// TwinCAT 3 PLC project CamerasTCP_Drivers
// ProgramVersion: 3.1.4026.19
// libraries:
//   AI Codes And Validation, * (Marden Edwards)
//   Tc2_SerialCom, * (Beckhoff Automation GmbH)
//   Tc2_Standard, * (Beckhoff Automation GmbH)
//   Tc2_System, * (Beckhoff Automation GmbH)
//   Tc2_TcpIp, * (Beckhoff Automation GmbH)
//   Tc2_Utilities, * (Beckhoff Automation GmbH)
//   TcUnit, * (www.tcunit.org)
// project tree:
//   DUTs/ E_TCPIP_RequescCommand.TcDUT, E_TCPIP_SEND_STATE.TcDUT, E_TCPIP_StateWP.TcDUT
//   DUTs/METS/ADS Symobol/ E_SYMBOL_AccessState.TcDUT, E_SYMBOL_AdsStates.TcDUT, ST_SYMBOL_AddressInfo.TcDUT
//   DUTs/METS/AI Codes And Validation/ E_CodeAI.TcDUT, E_CodeAIType.TcDUT (not stored), E_CodeType.TcDUT, ST_CodeInfo.TcDUT, ST_CodeValidation.TcDUT, ST_RejectItems.TcDUT, ST_RejectReasonsForCase.TcDUT, ST_RejectReasonsForOuter.TcDUT, ST_RejectReasonsForPack.TcDUT
//   DUTs/METS/AI Codes And Validation/GS1_Standard/ E_GS1_CodeAIType.TcDUT, E_GS1_CodeLvl.TcDUT, ST_GS1_AI_Attributs.TcDUT, ST_GS1_AI_Definition.TcDUT, ST_GS1_CodeInfo.TcDUT, ST_GS1_CodeValidation.TcDUT, ST_GS1_Decode_AI.TcDUT
//   DUTs/METS/Alarms/ E_MessageID.TcDUT (not stored), E_MessageType.TcDUT, ST_AlarmDB.TcDUT, ST_Alarms.TcDUT, ST_AlarmSettings.TcDUT, ST_AlarmsTable.TcDUT, ST_AlarmStatus.TcDUT, ST_ALARM_Aux.TcDUT (not stored)
//   DUTs/METS/Aliases/ T_CAC_Filename.TcDUT, T_CASE_Barcode.TcDUT, T_Char.TcDUT, T_CHM_Filename.TcDUT, T_CodeBATCH.TcDUT, T_CodeBRAND.TcDUT, T_CodeCRYPTO.TcDUT, T_CodeGTIN.TcDUT, T_CodeMRP.TcDUT, T_CodePIT.TcDUT, T_CodePO.TcDUT, T_CodePRODUCEDATE.TcDUT, T_CodeRSKU.TcDUT, T_CodeURL.TcDUT, T_DB_LongSTRING.TcDUT, T_FileExtension.TcDUT, T_FolderName.TcDUT, T_FolderPath.TcDUT, T_FSS_RejecCode.TcDUT, T_HMI_PACK_Barcode.TcDUT, T_ISO8601Time.TcDUT, T_LongSTRING.TcDUT, T_OAC_Filename.TcDUT, T_OCV_Filename.TcDUT, T_OHM_Filename.TcDUT, T_OUTER_Barcode.TcDUT, T_PACK_Barcode.TcDUT, T_PCM_Filename.TcDUT, T_PositiveDINT.TcDUT, T_PositiveINT.TcDUT, T_ProductDescription.TcDUT, T_RejectCode.TcDUT, T_TimeLog.TcDUT
//   DUTs/METS/Case/CAC/ E_CAC_State.TcDUT, ST_CAC_Data.TcDUT
//   DUTs/METS/Case/CHM/CHM Data Structure/GenericHierarchy/Case Item Structures/ ST_CaseContent.TcDUT, ST_CaseIdentity.TcDUT, ST_CaseItem.TcDUT
//   DUTs/METS/Case/CHM/CHM Data Structure/GenericHierarchy/Outer Item Structures/ ST_OuterContent.TcDUT, ST_OuterIdentity.TcDUT, ST_OuterItem.TcDUT
//   DUTs/METS/Case/CHM/CHM Data Structure/GenericHierarchy/Pack Item Structures/ ST_PackIdentity.TcDUT, ST_PackItem.TcDUT
//   DUTs/METS/Case/CHM/CHM Data Structure/GenericHierarchy/ ST_DefaultIdentity.TcDUT
//   DUTs/METS/Case/CHM/CHM Data Structure/ ST_Attributes.TcDUT, ST_CHM_GenericHierarchy.TcDUT (excluded from build), ST_GenericHierarchy.TcDUT, ST_MessageHeader.TcDUT
//   DUTs/METS/Case/CHM/ E_CHM_GeneratorState.TcDUT, E_CHM_State.TcDUT, E_CHM_WriteMode.TcDUT (excluded from build), ST_CHM_Data.TcDUT
//   DUTs/METS/Case/ E_CASE_State.TcDUT, ST_CasePackerInfo.TcDUT, ST_CASE_CaseQueue.TcDUT, ST_CASE_DefferOuter.TcDUT, ST_CASE_InfeedQueue.TcDUT, ST_CASE_OperationData.TcDUT (not stored)
//   DUTs/METS/Case/ORCA/ E_ORCA_State.TcDUT, ST_ORCA_BrandInfo.TcDUT, ST_ORCA_Data.TcDUT, ST_ORCA_Outers.TcDUT, ST_ORCA_ProductInfo.TcDUT, ST_ORCA_SiteInfo.TcDUT
//   DUTs/METS/Device/CX Unit/Device/ E_CX_DeviceState.TcDUT
//   DUTs/METS/Device/CX Unit/EtherCAT/ E_CX_EtherCATState.TcDUT (not stored), ST_CX_EtherCATDeviceState.TcDUT, ST_CX_EtherCATMasterPNetState.TcDUT, ST_CX_EtherCATMasterState.TcDUT
//   DUTs/METS/Device/CX Unit/EtherCAT/Terminal FBs/EBUS/ ST_EBUS_AnalogueDataIn.TcDUT, ST_EBUS_EtherCATState.TcDUT
//   DUTs/METS/Device/CX Unit/EtherCAT/Terminal FBs/KBUS/ E_KBUS_RegisterAccessState.TcDUT, ST_KBUS_AnalogueDataIn.TcDUT, ST_KBUS_AnalogueDataOut.TcDUT, ST_KBUS_KL1501DataIn.TcDUT, ST_KBUS_KL1501DataOut.TcDUT, ST_KBUS_KL5001Config.TcDUT
//   DUTs/METS/Device/CX Unit/EtherCAT/Terminal FBs/ ST_EtherCATSlaveInfo.TcDUT, ST_EtherCATStatus.TcDUT
//   DUTs/METS/Device/CX Unit/Network/ E_CX_NetworkInfoState.TcDUT, E_CX_SetAMSNetIDState.TcDUT, ST_CX_AdapterInfo.TcDUT, ST_CX_NetworkInfo.TcDUT
//   DUTs/METS/Device/CX Unit/NOVRAM/ E_CX_NVDataCtrlState.TcDUT, E_CX_NVDataOpMode.TcDUT (not stored), E_CX_NVXMLState.TcDUT (not stored), ST_CX_AMSAddress.TcDUT, ST_CX_EL6080DataIn.TcDUT, ST_CX_EL6080DataOut.TcDUT, ST_CX_NVDataBlock.TcDUT
//   DUTs/METS/Device/CX Unit/System/ E_CX_HWType.TcDUT, E_CX_State.TcDUT (not stored)
//   DUTs/METS/Device/Cylinders/ E_CYLINDER_Name.TcDUT (not stored), E_CYLINDER_Position.TcDUT, ST_CYLINDER_Config.TcDUT (not stored), ST_CYLINDER_Control.TcDUT, ST_CYLINDER_IN.TcDUT, ST_CYLINDER_OUT.TcDUT, ST_CYLINDER_Status.TcDUT, ST_CYLINDER_TagID.TcDUT
//   DUTs/METS/Device/DB/ E_DB_ScanState.TcDUT (not stored), ST_DB_CACDataCtrl.TcDUT (not stored), ST_DB_OACDataCtrl.TcDUT, ST_DB_OCVDataCtrl.TcDUT
//   DUTs/METS/Device/DB/OLD/ ST_DBResult.TcDUT (excluded from build), ST_DB_CACCheckCtrl.TcDUT (excluded from build), ST_DB_Config.TcDUT, ST_DB_OACCheckCtrl.TcDUT (excluded from build), ST_DB_OCVCheckCtrl.TcDUT (excluded from build), ST_DB_PcvCheckCtrl.TcDUT (excluded from build), ST_DB_ReportDBCtrl.TcDUT, ST_DB_ReportResult.TcDUT
//   DUTs/METS/Device/Drive/Analog/Config/ ST_AnalogDrive.TcDUT
//   DUTs/METS/Device/Drive/Analog/ ST_DriveCtrl.TcDUT, ST_PhtcCtrl.TcDUT (excluded from build)
//   DUTs/METS/Device/Drive/MC2/Axis Control/ E_AXIS_MotionType.TcDUT (not stored), ST_AXIS_Control.TcDUT, ST_AXIS_IN.TcDUT, ST_AXIS_OUT.TcDUT, ST_AXIS_Status.TcDUT
//   DUTs/METS/Device/Drive/MC2/Config/ ST_AXIS_Config.TcDUT
//   DUTs/METS/Device/Drive/MC2/EtherCAT/AX5000 FBs/ ST_AX5000_TouchProbe.TcDUT
//   DUTs/METS/Device/Drive/MC2/EtherCAT/Encoder FBs/ ST_DeviceAddress.TcDUT
//   DUTs/METS/Device/Drive/MC2/ E_MC_Name.TcDUT (not stored)
//   DUTs/METS/Device/Drive/MC2/NC Axis/Cam/ E_CAM_Update.TcDUT (not stored)
//   DUTs/METS/Device/Drive/MC2/NC Axis/ E_AXIS_CtrlState.TcDUT, E_TORQUE_Scaling.TcDUT, ST_AxisCtrlRamps.TcDUT, ST_DriveStatus.TcDUT, ST_LatchPosBuffer.TcDUT, ST_NC_EncDataIn.TcDUT, ST_NC_EncDataOut.TcDUT
//   DUTs/METS/Device/Drive/MC2/TempAxis/ ST_AxisHomeStruct.TcDUT (excluded from build), ST_AxisMotionStruct.TcDUT (excluded from build)
//   DUTs/METS/Device/Drive/Profinet/Config/ ST_ProfinetDrive.TcDUT, ST_ProfinetMasterConfig.TcDUT
//   DUTs/METS/Device/Drive/Profinet/ E_DRIVE_Name.TcDUT, ST_PNetMasterStatus.TcDUT
//   DUTs/METS/Device/Drive/Profinet/Parameters/ ST_DataPntAdr.TcDUT, ST_KeyPadDisplay.TcDUT, ST_Parameter.TcDUT, ST_ParameterControl.TcDUT, ST_Parameters.TcDUT, ST_Value.TcDUT
//   DUTs/METS/Device/Drive/Profinet/_G120/Drives/ E_DRIVE_DataType.TcDUT, ST_DRIVE_INPUT.TcDUT, ST_DRIVE_OUTPUT.TcDUT, ST_DRIVE_STATUS.TcDUT, ST_G120_ExtendedIn.TcDUT, ST_G120_ExtendedOut.TcDUT, ST_G120_IN.TcDUT, ST_G120_OUT.TcDUT (not stored), ST_G120_Status.TcDUT
//   DUTs/METS/Device/Drive/Profinet/_G120/ ST_G120_Control.TcDUT
//   DUTs/METS/Device/Encoders/CAMS/ ST_AFS60_Cam.TcDUT, ST_AFS60_CamHMi.TcDUT, ST_AFS60_Config.TcDUT, ST_AFS60_Status.TcDUT
//   DUTs/METS/Device/Encoders/ E_ENOCDER_Name.TcDUT (not stored), ST_ENCODER_IN.TcDUT, ST_ENCODER_OUT.TcDUT, ST_ENCODER_Status.TcDUT
//   DUTs/METS/Device/IO2 Controls/ E_IO2_InputSource.TcDUT, E_IO2_Type.TcDUT, ST_IO2_Diagnostic.TcDUT, ST_IO2_InputPLC.TcDUT, ST_IO2_OutputPLC.TcDUT
//   DUTs/METS/Device/IO2 Controls/Input Ctrl/ ST_IO2_DoubleInputCtrl.TcDUT, ST_IO2_DoubleInputLockedCtrl.TcDUT, ST_IO2_SingleInputCtrl.TcDUT, ST_IO2_SingleInputLockedCtrl.TcDUT
//   DUTs/METS/Device/IO2 Controls/Outpout Ctrl/ ST_IO2_OutputCtrl.TcDUT
//   DUTs/METS/Device/Printers/ E_PRINTER_Name.TcDUT (not stored), E_PRINTER_State.TcDUT, ST_PRINTER_Config.TcDUT, ST_PRINTER_IN.TcDUT, ST_PRINTER_OUT.TcDUT, ST_PRINTER_Status.TcDUT
//   DUTs/METS/Device/Scanner/ E_ClientSteps.TcDUT (not stored), E_DataExchaSteps.TcDUT (not stored), E_SCANNER_CodeType.TcDUT, E_SCANNER_DeviceType.TcDUT, E_SCANNER_Name.TcDUT (not stored), E_SCANNER_State.TcDUT, E_SCANNER_Vendor.TcDUT, ST_SCANNER.TcDUT, ST_SCANNER_ApplicationIdentifier.TcDUT, ST_SCANNER_CameraMap.TcDUT, ST_SCANNER_CodeData.TcDUT, ST_SCANNER_Config.TcDUT, ST_SCANNER_Evaluation.TcDUT, ST_SCANNER_ImageData.TcDUT, ST_SCANNER_ManualCtrl.TcDUT, ST_SCANNER_OpState.TcDUT, ST_SCANNER_Options.TcDUT, ST_SCANNER_Performance.TcDUT, ST_SCANNER_Statistics.TcDUT, ST_SCANNER_TriggerID.TcDUT
//   DUTs/METS/Device/Scanner/Hand Scanner/ E_ConnectSteps.TcDUT (not stored), E_DataSequence.TcDUT, E_SCANNER_Baudrate.TcDUT (not stored), ST_SCANNER_HoneywellConfig.TcDUT, ST_SCANNER_HoneywellCtrl.TcDUT, ST_SCANNER_HoneywellStatus.TcDUT, ST_SCANNER_HostAck.TcDUT, ST_SCANNER_USBConfig.TcDUT
//   DUTs/METS/Device/Scanner/NewModel/ ST_SCANNER_Configuration.TcDUT (not stored), ST_SCANNER_Ctrl.TcDUT, ST_SCANNER_CtrlMapping.TcDUT (not stored), ST_SCANNER_CtrlOptions.TcDUT (excluded from build), ST_SCANNER_IN.TcDUT, ST_SCANNER_ManualStatus.TcDUT (not stored), ST_SCANNER_OUT.TcDUT (not stored), ST_SCANNER_Status.TcDUT (not stored)
//   DUTs/METS/Files/ E_FILE_CtrlState.TcDUT, E_FILE_DeleteOldFilesState.TcDUT, E_FILE_State.TcDUT, ST_FILE_WriteFileStatistic.TcDUT
//   DUTs/METS/HMI/Device Manual Control/ ST_HMI_AxisCtrl.TcDUT, ST_HMI_CylinderCtrl.TcDUT (not stored), ST_HMI_G120Ctrl.TcDUT, ST_HMI_PrinterCtrl.TcDUT
//   DUTs/METS/HMI/Device Status/ E_HMI_DriveStatus.TcDUT, ST_HMI_AxisStatus.TcDUT, ST_HMI_CylinderStatus.TcDUT, ST_HMI_G120Status.TcDUT (not stored), ST_HMI_HoneywellStatus.TcDUT, ST_HMI_PrinterStatus.TcDUT
//   DUTs/METS/HMI/HMIQueue/ ST_HMI_CAC_Data.TcDUT, ST_HMI_CaseRejectCode.TcDUT (not stored), ST_HMI_CaseVerifiedCode.TcDUT, ST_HMI_CASE_CaseQueue.TcDUT, ST_HMI_InfeedQueue.TcDUT (not stored), ST_HMI_OAC_Data.TcDUT, ST_HMI_OCV_Data.TcDUT, ST_HMI_OuterStatus.TcDUT, ST_HMI_PACK_BufferStatus.TcDUT (not stored), ST_HMI_PLAS_Queue.TcDUT
//   DUTs/METS/HMI/ ST_HMI_BarGraph.TcDUT (not stored), ST_HMI_Buttons.TcDUT, ST_HMI_CSVStoreTable.TcDUT (not stored), ST_HMI_StationStatus.TcDUT, ST_HMI_Visualisation.TcDUT
//   DUTs/METS/KPI/ ST_KPI_CasePackerSignals.TcDUT, ST_KPI_CodePos.TcDUT, ST_KPI_InspectionEfficency.TcDUT, ST_KPI_ItemsProduced.TcDUT, ST_KPI_OCVFile.TcDUT, ST_KPI_OutersProcessing.TcDUT, ST_KPI_OutersProduced.TcDUT
//   DUTs/METS/LogData/ E_LOG_Handler.TcDUT, ST_LOG_Alarms.TcDUT, ST_LOG_EventData.TcDUT, ST_LOG_FileWriteError.TcDUT, ST_LOG_MachineState.TcDUT, ST_LOG_RejectReasons.TcDUT (not stored), ST_LOG_WriteImageData.TcDUT
//   DUTs/METS/NV Data/ ST_NOVRAM_METS_Cameras.TcDUT, ST_NOVRAM_METS_CaseInspactionLog.TcDUT, ST_NOVRAM_METS_DualInputs.TcDUT, ST_NOVRAM_METS_EventCounters.TcDUT (not stored), ST_NOVRAM_METS_Inspection.TcDUT
//   DUTs/METS/Outers/ E_OUTER_AgrregationState.TcDUT, E_OUTER_State.TcDUT, ST_OUTER_Status.TcDUT
//   DUTs/METS/Outers/OAC/ E_OAC_State.TcDUT, ST_OAC_Data.TcDUT
//   DUTs/METS/Outers/SFLX/ E_SIDEFLEX_UnitType.TcDUT, ST_SIDEFLEX_Offset.TcDUT, ST_SIDEFLEX_ProcessData.TcDUT
//   DUTs/METS/Packs/ E_OCV_CheckMode.TcDUT, E_OCV_State.TcDUT, E_PACK_FilledInStatus.TcDUT, E_PACK_ReadStep.TcDUT, E_PACK_State.TcDUT, ST_PACK_CodeBuffer.TcDUT, ST_PACK_CodeStatus.TcDUT, ST_PACK_ConfirmationQueue.TcDUT, ST_PACK_Data.TcDUT, ST_PACK_DuplicatesCheck.TcDUT (not stored), ST_PACK_InfeedQueue.TcDUT, ST_PACK_InTransferQueue.TcDUT, ST_PACK_LastFilledCodes.TcDUT (not stored), ST_PACK_TriggerOffset.TcDUT
//   DUTs/METS/Packs/_Lab/ ST_LAB_OuterData_1.TcDUT, ST_LAB_PackData_1.TcDUT
//   DUTs/METS/PCM/ E_PCM_State.TcDUT (not stored), ST_PCM_Data.TcDUT (not stored), ST_PCM_Status.TcDUT
//   DUTs/METS/PCM/PCM_Hierarchy/ProductInformation/Product/ ST_HierarchyData.TcDUT, ST_HierarchyDataList.TcDUT (not stored)
//   DUTs/METS/PCM/PCM_Hierarchy/ProductInformation/Settings/ ST_ToleranceThresholdCS.TcDUT, ST_ToleranceThresholdOUT.TcDUT, ST_ToleranceThresholdPK.TcDUT (not stored)
//   DUTs/METS/PCM/PCM_Hierarchy/ProductInformation/ ST_PCMProduct.TcDUT (not stored), ST_PCMSettings.TcDUT (not stored)
//   DUTs/METS/PCM/PCM_Hierarchy/ ST_PCMMessageHeader.TcDUT (not stored), ST_ProductInformation.TcDUT (not stored)
//   DUTs/METS/String Processing/ E_STRING_ExtrMode.TcDUT (not stored)
//   DUTs/METS/System/ E_SYSTEM_CTState.TcDUT, E_SYSTEM_HandScannerBaudrate.TcDUT, E_SYSTEM_ItemType.TcDUT, E_SYSTEM_MachineState.TcDUT, E_SYSTEM_MaintainFolders.TcDUT, E_SYSTEM_OSType.TcDUT, ST_SYSTEM_Config.TcDUT, ST_SYSTEM_DateTime.TcDUT, ST_SYSTEM_DeviceState.TcDUT, ST_SYSTEM_Door.TcDUT, ST_SYSTEM_MachineID.TcDUT (not stored), ST_SYSTEM_MachineMode.TcDUT, ST_SYSTEM_MachineState.TcDUT, ST_SYSTEM_ProductionLine.TcDUT, ST_SYSTEM_SafetyStatus.TcDUT, ST_SYSTEM_SoftwareVersion.TcDUT
//   DUTs/METS/System/Status/ ST_SYSTEM_ArchiveDBStatus.TcDUT (not stored), ST_SYSTEM_BridgeStatus.TcDUT, ST_SYSTEM_LoggerStatus.TcDUT (not stored), ST_SYSTEM_MachineStatus.TcDUT, ST_SYSTEM_ReportingDBStatus.TcDUT
//   DUTs/METS/System/System Modes/ E_SYSTEM_AutomationMode.TcDUT (not stored), E_SYSTEM_OuterAggregationMode.TcDUT (not stored), E_SYSTEM_PackAggregationMode.TcDUT
//   DUTs/METS/TCPIP Address/ E_TCPIP_State_1.TcDUT, ST_TCPIP_AddressPort.TcDUT
//   DUTs/METS/XML Processing/ E_XML_CtrlState.TcDUT, E_XML_GeneratorState.TcDUT, E_XML_WritingMode.TcDUT
//   DUTs/METS/_StationOperational/C715 Tempalate Example/ E_04_ElevatorState_C715.TcDUT, E_Axis_C715.TcDUT, E_Cylinder_C715.TcDUT, ST_04_ElevatorSeq_C715.TcDUT, ST_BundleTrackingRegister_C715.TcDUT, ST_CommonStationConfig_C715.TcDUT (not stored)
//   DUTs/METS/_StationOperational/ E_00_StationStateTemplate.TcDUT, ST_00_StationStructTemplate.TcDUT
//   DUTs/METS/_StationOperational/Manual Machine/ E_OuterPrintStationState.TcDUT, ST_OuterPrintStationStruct.TcDUT
//   DUTs/METS/_StationOperational/SeqCtrl/ ST_STATION_Requests.TcDUT, ST_STATION_Status.TcDUT
//   DUTs/Test_DUTs/ ST_DuplicateInfo.TcDUT, ST_FBinside.TcDUT, ST_LAB_CaseData.TcDUT, ST_LAB_OuterData.TcDUT, ST_LAB_PackData.TcDUT
//   GVLs/ CodeAI.TcGVL, gConstants.TcGVL, GVL.TcGVL, GVL_HIKROBOT_COMMANDS.TcGVL, GVL_test.TcGVL
//   / PlcTask.TcTTO, TcUnit_Task.TcTTO
//   POUs/FBReferenceTest/ FB_TimersTEST.TcPOU, PRG_Reference_POU.TcPOU
//   POUs/FinaliseCaseData/ FB_CASE_DuplicatCheck.TcPOU, FB_CASE_DuplicateUpdateToDB.TcPOU, FB_CASE_FinaliseData.TcPOU, FB_CASE_InitialiseData.TcPOU, FB_CASE_MovePackerToCase.TcPOU, FB_CASE_ValidateContent.TcPOU
//   POUs/ PRG_TEST.TcPOU
//   POUs/TcUnit/FB_CASE_DuplicatCheckTests/ FB_CASE_DuplicatCheckTests.TcPOU, PRG_CASE_DuplicatCheckManual.TcPOU
//   POUs/TcUnit/FB_CASE_DuplicateUpdateToDBTests/ PRG_CASE_DuplicateUpdateToDBManual.TcPOU, FB_CASE_DuplicateUpdateToDBTests.TcPOU
//   POUs/TcUnit/FB_CASE_ValidateContentTests/ FB_CASE_ValidateContentTests.TcPOU, PRG_CASE_ValidateContentManual.TcPOU
//   POUs/TcUnit/FB_CASE_InitialiseData/ FB_CASE_InitialiseDataTests.TcPOU, PRG_CASE_InitialiseDataManual.TcPOU
//   POUs/TcUnit/FB_CASE_FinaliseDataTests/ FB_CASE_FinaliseDataTests.TcPOU, PRG_CASE_FinaliseDataManual.TcPOU
//   POUs/TcUnit/F_CODE_GetItemAITests/ PRG_CODE_GetItemAIManual.TcPOU
//   POUs/_Utilites/Addtionals/ FB_PulseGenerator_Sync.TcPOU, PRG_ButtonsHandler.TcPOU
//   POUs/_Utilites/CAMERAS/ FB_SCANNER_HikrobotEXT.TcPOU, F_CREATE_MESSAGE.TcPOU
//   POUs/_Utilites/METS/Common LIB/08_SOFTWARE LIB/AI Codes And Validation FBs/ FB_CODE_ClearCodeInfo.TcPOU, FB_CODE_ValidateExplicitCode.TcPOU (not stored), F_CODE_AssignValToStringWithPrefix.TcPOU, F_CODE_GetItemAI.TcPOU (not stored)
//   POUs/_Utilites/METS/Common LIB/08_SOFTWARE LIB/AI GS1 Codes And Validation FBs/ FB_GS1_ClearCodeInfo.TcPOU, FB_GS1_ValidateExplicitCode.TcPOU, F_GS1_GetItem.TcPOU
//   POUs/_Utilites/METS/Concat Function/ F_CONCAT3.TcPOU, F_CONCAT4.TcPOU, F_CONCAT5.TcPOU, F_CONCAT6.TcPOU, F_CONCAT7.TcPOU, F_CONCAT8.TcPOU, F_CONCAT9.TcPOU
//   POUs/_Utilites/METS/ FB_ExtractString.TcPOU (not stored), F_CASE_GetSKUFromHex.TcPOU, F_CODE_BATSerializator.TcPOU (not stored), F_CODE_GetItem.TcPOU, F_FiltredSetBitState16.TcPOU, F_InvalidateASCIIChar.TcPOU, F_SafeDIV.TcPOU, F_StringAddPrefix.TcPOU (not stored), F_StringWildcard.TcPOU, F_SYSTEM_SystemTimeAsISO8601.TcPOU, F_SYSTEM_SystemTimeOffsetToHHMM.TcPOU, F_ZeroPadString.TcPOU
//   POUs/_Utilites/TCP_FB/ FB_ReceiveString.TcPOU, FB_TCP_ClientPortCtrl.TcPOU
//   POUs/_Utilites/Tests/ FB_FIND_OuterDuplicates.TcPOU, FB_FIND_OuterDuplicatesPiotr.TcPOU, FB_FIND_OuterDuplicatesPiotrAI.TcPOU, IO_logic.TcPOU, Outer_IN_Case_Duplicat.TcPOU, PRG_TestCamera.TcPOU

CONFIGURATION CamerasTCP_Drivers
    RESOURCE PLC ON TwinCAT3
        TASK PlcTask(INTERVAL := T#20ms, PRIORITY := 20);
        TASK TcUnit_Task(INTERVAL := T#1ms, PRIORITY := 25);
        PROGRAM PRG_TEST WITH TcUnit_Task : PRG_TEST;
    END_RESOURCE
END_CONFIGURATION

// ---- DUTs/E_TCPIP_RequescCommand.TcDUT
{attribute 'qualified_only'}
{attribute 'strict'}
{attribute 'to_string'}
TYPE E_TCPIP_RequescCommand :
(
	NONE,					(* No request to send *)
	SetRunMode,				(* Set run mode, 0 - Normal, 1 - Raw, 2 - Test *)
	SetAcq,					(* Set acquisition mode, 0 - Stop acq, 1 - Start acq *)
	GetUserCur,
	HeartbeatCheck,		
	SetAquisitonModeON,
	SetAquisitionModeOFF,
	WrongReply	
);
END_TYPE

// ---- DUTs/E_TCPIP_SEND_STATE.TcDUT
{attribute 'qualified_only'}
{attribute 'strict'}
{attribute 'to_string'}
TYPE E_TCPIP_SEND_STATE :
(
	WAITING,
	SEND,
	RECEIVE,
	DONE,
	CONN_RESET,
	HEARTBEAT_CHECK
);
END_TYPE

// ---- DUTs/E_TCPIP_StateWP.TcDUT
{attribute 'qualified_only'}
{attribute 'strict'}
{attribute 'to_string'}
TYPE E_TCPIP_StateWP :
(
	E_TCPIP_IDLE,
	E_TCPIP_CONNECT,
	E_TCPIP_SEND,
	E_TCPIP_RECEIVE,
	E_TCPIP_DISCONNECT,
	E_TCPIP_CLOSEALL,
	E_TCPIP_DONE
);
END_TYPE

// ---- DUTs/METS/ADS Symobol/E_SYMBOL_AccessState.TcDUT
TYPE E_SYMBOL_AccessState :
(
	E_SYMBOL_IDLE,
	E_SYMBOL_GETSYMBOLINFO,
	E_SYMBOL_READDATA,
	E_SYMBOL_WRITEDATA,
	E_SYMBOL_DONE
);
END_TYPE

// ---- DUTs/METS/ADS Symobol/E_SYMBOL_AdsStates.TcDUT
TYPE E_SYMBOL_AdsStates :
(
	ADSSTATES_INVALID :=0,
	ADSSTATES_IDLE :=1,
	ADSSTATES_RESET :=2,
	ADSSTATES_INIT :=3,
	ADSSTATES_START :=4,
	ADSSTATES_RUN :=5,
	ADSSTATES_STOP :=6,
	ADSSTATES_SAVECFG :=7,
	ADSSTATES_LOADCFG :=8,
	ADSSTATES_POWERFAILURE :=9,
	ADSSTATES_POWERGOOD :=10,
	ADSSTATES_ERROR :=11
);
END_TYPE

// ---- DUTs/METS/ADS Symobol/ST_SYMBOL_AddressInfo.TcDUT
TYPE ST_SYMBOL_AddressInfo :	(* 8 bytes *)
STRUCT
	pSymAddr	: 	DWORD;
	nSymSize	:	UDINT;
END_STRUCT
END_TYPE

// ---- DUTs/METS/AI Codes And Validation/E_CodeAI.TcDUT
{attribute 'qualified_only'}
TYPE E_CodeAI :
(
	GTIN 			:= 1,
	BATCH 			:= 10,
	SERIAL			:= 21,
	PO				:= 91,
	BRANDSPEC		:= 92,
	CRYPTO			:= 93,
	PRODDATE		:= 94,
	RSKU 			:= 240,
	MRP				:= 8005,
	USERFIELD		:= 999
);
END_TYPE

// ---- DUTs/METS/AI Codes And Validation/E_CodeType.TcDUT
TYPE E_CodeType :
(
	E_NONE,
	E_PACK,
	E_INTERIM,
	E_OUTER,
	E_CASE

);
END_TYPE

// ---- DUTs/METS/AI Codes And Validation/GS1_Standard/E_GS1_CodeAIType.TcDUT
TYPE E_GS1_CodeAIType :
(
	GS1_00		:= 0,		(*GS1 Not defined*)
	GS1_01		 :=1,		(***********Global Trade Item Number (GTIN)	N2+N14*************)
	GS1_10		:=10,		(***********Batch or lot number	N2+X..20*************)
	GS1_11		:=11,		(***********Production date (YYMMDD)		N2+N6*************)
	GS1_15		:=15,		(***********Best before date (YYMMDD)			N2+N6*************)
	GS1_17		:=17,		(***********Expiration date (YYMMDD)		N2+N6*************)
	GS1_21		:=21,		(***********Serial number		N2+X..20*************)
	GS1_240		:=240,	(***********Additional product identification assigned by the manufacturer	N3+X..30*************)
	GS1_8005		:=8005,	(***********Price per unit of measure	N4+N6*************)
	GS1_8006		:=8006,	(***********Identification of an individual trade item piece	N4+N14+N2+N2*************)
	GS1_8008		:=8008,	(***********Date and time of production		N4+N8+N..4*************)
	GS1_91		:=91,		(***********Company internal information	N2+X..90*************)
	GS1_92		:=92,		(***********Company internal information	N2+X..90*************)
	GS1_93		:=93,		(***********Company internal information	N2+X..90*************)
	GS1_94		:=94,		(***********Company internal information	N2+X..90*************)
	NON_GS1_01		:=10001,	(***********Non GS1 - user defined		X..255*************)
	NON_GS1_02		:=10002,	(***********Non GS1 - user defined		X..255*************)
	NON_GS1_03		:=10003,	(***********Non GS1 - user defined		X..255*************)
	NON_GS1_04		:=10004,	(***********Non GS1 - user defined		X..255*************)
	NON_GS1_05		:=10005,	(***********Non GS1 - user defined		X..255*************)
	NON_GS1_06		:=10006,	(***********Non GS1 - user defined		X..255*************)
	NON_GS1_07		:=10007,	(***********Non GS1 - user defined		X..255*************)
	NON_GS1_08		:=10008,	(***********Non GS1 - user defined		X..255*************)
	NON_GS1_09		:=10009,	(***********Non GS1 - user defined		X..255*************)
	NON_GS1_10		:=10010	(***********Non GS1 - user defined		X..255*************)
);
END_TYPE

// ---- DUTs/METS/AI Codes And Validation/GS1_Standard/E_GS1_CodeLvl.TcDUT
TYPE E_GS1_CodeLvl :
(
	E_LVL_NONE,
	E_LEVEL1,
	E_LEVEL2,
	E_LEVEL3
);
END_TYPE

// ---- DUTs/METS/AI Codes And Validation/GS1_Standard/ST_GS1_AI_Attributs.TcDUT
TYPE ST_GS1_AI_Attributs :
STRUCT
	sDataField 	: T_MaxString;
	bDataChanged	: BOOL;
	sAI_Id		: STRING(5);
	eGS1_AI		: E_GS1_CodeAIType;
	bFixed		: BOOL;
	nLength		: UINT;
END_STRUCT
END_TYPE

// ---- DUTs/METS/AI Codes And Validation/GS1_Standard/ST_GS1_AI_Definition.TcDUT
TYPE ST_GS1_AI_Definition :
STRUCT
	sDotCode_CI	: STRING(3) := ']j';			(* GS1 marker (FNC1 Carrier Identifiers for DataMatrix barcode *)
	sDMC_CI		: STRING(3) := ']d2';			(* GS1 marker (FNC1 Carrier Identifiers for DataMatrix barcode *)
	sCode128_CI	: STRING(3) := ']c1';			(* GS1 marker (FNC1 Carrier Identifiers for Code128 barcode *)
	stAI_01_Lvl1	: ST_GS1_AI_Attributs := (sAI_Id:='01', eGS1_AI:=GS1_01, bFixed:= TRUE, nLength:=14);	(***********N2+N14*************)
	stAI_01_Lvl2	: ST_GS1_AI_Attributs := (sAI_Id:='01', eGS1_AI:=GS1_01, bFixed:= TRUE, nLength:=14);	(***********N2+N14*************)
	stAI_01_Lvl3	: ST_GS1_AI_Attributs := (sAI_Id:='01', eGS1_AI:=GS1_01, bFixed:= TRUE, nLength:=14);	(***********N2+N14*************)
	stAI_10		: ST_GS1_AI_Attributs := (sAI_Id:='10', eGS1_AI:=GS1_10, bFixed:= FALSE, nLength:=20);	(***********N2+X..20*************)
	stAI_11		: ST_GS1_AI_Attributs := (sAI_Id:='11', eGS1_AI:=GS1_11, bFixed:= TRUE, nLength:=6);	(***********N2+N6*************)
	stAI_15		: ST_GS1_AI_Attributs := (sAI_Id:='15', eGS1_AI:=GS1_15, bFixed:= TRUE, nLength:=6);	(***********N2+N6*************)
	stAI_17		: ST_GS1_AI_Attributs := (sAI_Id:='17', eGS1_AI:=GS1_17, bFixed:= TRUE, nLength:=6);	(***********N2+N6*************)
	stAI_21		: ST_GS1_AI_Attributs := (sAI_Id:='21', eGS1_AI:=GS1_21, bFixed:= FALSE, nLength:=20);	(***********N2+X..20*************)
	stAI_240		: ST_GS1_AI_Attributs := (sAI_Id:='240', eGS1_AI:=GS1_240, bFixed:= FALSE, nLength:=30);		(***********N3+X..30*************)
	stAI_8005		: ST_GS1_AI_Attributs := (sAI_Id:='8005', eGS1_AI:=GS1_8005, bFixed:= TRUE, nLength:=6);		(***********N4+N6*************)
	stAI_8006		: ST_GS1_AI_Attributs := (sAI_Id:='8006', eGS1_AI:=GS1_8006, bFixed:= TRUE, nLength:=18);	(***********N4+N14+N2+N2*************)
	stAI_8008		: ST_GS1_AI_Attributs := (sAI_Id:='8008', eGS1_AI:=GS1_8008, bFixed:= TRUE, nLength:=12);	(***********N4+N8+N..4*************)
	stAI_91		: ST_GS1_AI_Attributs := (sAI_Id:='91', eGS1_AI:=GS1_91, bFixed:= FALSE, nLength:=90);		(***********N2+X..90*************)
	stAI_92		: ST_GS1_AI_Attributs := (sAI_Id:='92', eGS1_AI:=GS1_92, bFixed:= FALSE, nLength:=90);		(***********N2+X..90*************)
	stAI_93		: ST_GS1_AI_Attributs := (sAI_Id:='93', eGS1_AI:=GS1_93, bFixed:= FALSE, nLength:=90);		(***********N2+X..90*************)
	stAI_94		: ST_GS1_AI_Attributs := (sAI_Id:='94', eGS1_AI:=GS1_94, bFixed:= FALSE, nLength:=90);		(***********N2+X..90*************)

	stNON_GS1_01		: ST_GS1_AI_Attributs := (sAI_Id:='10001', eGS1_AI:=NON_GS1_01, bFixed:= FALSE, nLength:=255);		(***********X..255*************)
	stNON_GS1_02		: ST_GS1_AI_Attributs := (sAI_Id:='10002', eGS1_AI:=NON_GS1_02, bFixed:= FALSE, nLength:=255);		(***********X..255*************)
	stNON_GS1_03		: ST_GS1_AI_Attributs := (sAI_Id:='10003', eGS1_AI:=NON_GS1_03, bFixed:= FALSE, nLength:=255);		(***********X..255*************)
	stNON_GS1_04		: ST_GS1_AI_Attributs := (sAI_Id:='10004', eGS1_AI:=NON_GS1_04, bFixed:= FALSE, nLength:=255);		(***********X..255*************)
	stNON_GS1_05		: ST_GS1_AI_Attributs := (sAI_Id:='10005', eGS1_AI:=NON_GS1_05, bFixed:= FALSE, nLength:=255);		(***********X..255*************)
	stNON_GS1_06		: ST_GS1_AI_Attributs := (sAI_Id:='10006', eGS1_AI:=NON_GS1_06, bFixed:= FALSE, nLength:=255);		(***********X..255*************)
	stNON_GS1_07		: ST_GS1_AI_Attributs := (sAI_Id:='10007', eGS1_AI:=NON_GS1_07, bFixed:= FALSE, nLength:=255);		(***********X..255*************)
	stNON_GS1_08		: ST_GS1_AI_Attributs := (sAI_Id:='10008', eGS1_AI:=NON_GS1_08, bFixed:= FALSE, nLength:=255);		(***********X..255*************)
	stNON_GS1_09		: ST_GS1_AI_Attributs := (sAI_Id:='10009', eGS1_AI:=NON_GS1_09, bFixed:= FALSE, nLength:=255);		(***********X..255*************)
	stNON_GS1_10		: ST_GS1_AI_Attributs := (sAI_Id:='10010', eGS1_AI:=NON_GS1_10, bFixed:= FALSE, nLength:=255);		(***********X..255*************)

END_STRUCT
END_TYPE

// ---- DUTs/METS/AI Codes And Validation/GS1_Standard/ST_GS1_CodeInfo.TcDUT
TYPE ST_GS1_CodeInfo :
STRUCT
	eCodeLvlType					:	E_GS1_CodeLvl;

	nMinLength					: 	INT;
	nEntireLength					:	INT;
	bValidateEntireLength			: 	BOOL;
	nNumberOfAIs					:	INT;

	stGS1_Field 					: ARRAY[1..cMAX_VALIDATION_ITEMS] OF 	ST_GS1_CodeValidation	;

	(*stGS1_Field01 				:	ST_GS1_CodeValidation	;
	stGS1_Field02 					:	ST_GS1_CodeValidation	;
	stGS1_Field03 					:	ST_GS1_CodeValidation	;
	stGS1_Field04 					:	ST_GS1_CodeValidation	;
	stGS1_Field05					:	ST_GS1_CodeValidation	;
	stGS1_Field06					:	ST_GS1_CodeValidation	;
	stGS1_Field07		 			:	ST_GS1_CodeValidation	;
	stGS1_Field08					:	ST_GS1_CodeValidation	;
	stGS1_Field09					:	ST_GS1_CodeValidation	;
	stGS1_Field10					:	ST_GS1_CodeValidation	;*)

END_STRUCT
END_TYPE

// ---- DUTs/METS/AI Codes And Validation/GS1_Standard/ST_GS1_CodeValidation.TcDUT
TYPE ST_GS1_CodeValidation :
STRUCT

	bValidate 			:	BOOL;
	sFieldName		:	STRING(15)	:='';

	sStartAI 			: 	STRING(6)		:= '';
	sEndAI 			: 	STRING(6) 	:= '';
	nCodeStartPos		:	INT;
	nCodeLength		:	INT;

	eGS1_AIType		: 	E_GS1_CodeAIType 	:= GS1_00;

(* If sStartAI is empty, then use nCodeStartPos, else find sStartAI in code for start position *)
(* If sEndAI is empty then use nCodeLength, else find sEndAI in code for end position*)

(*General Application Idendifiers (AI) Description:
	01:		GTIN
	10: 		Batch ID/WorkOrderID
	21: 		Serial Code
	91:		Production Order/WorkCenterID
	93:		Crypto
	240:		RSKU
*)

END_STRUCT
END_TYPE

// ---- DUTs/METS/AI Codes And Validation/GS1_Standard/ST_GS1_Decode_AI.TcDUT
TYPE ST_GS1_Decode_AI :
STRUCT
	sAI_Id		: STRING(5);
	bFixed		: BOOL;
	nLength		: UINT;
END_STRUCT
END_TYPE

// ---- DUTs/METS/AI Codes And Validation/ST_CodeInfo.TcDUT
TYPE ST_CodeInfo :
STRUCT
	eCodeType					:	E_CodeType;

	nMinLength					: 	INT;
	nEntireLength					:	INT;
	bValidateEntireLength			: 	BOOL;
	nNumberOfAIs					:	INT;

	stGTIN 						:	ST_CodeValidation	:=		(sFieldName :='GTIN',						bNameEditable := FALSE, 		nGS1_AI := 1);
	stBatchID 						:	ST_CodeValidation	:=		(sFieldName :='BatchID', 				bNameEditable := FALSE, 		nGS1_AI := 10);
	stSerialCode 					:	ST_CodeValidation	:=		(sFieldName :='SerialCode', 			bNameEditable := FALSE, 		nGS1_AI := 21);
	stProductionOrder 				:	ST_CodeValidation	:=		(sFieldName :='ProductionOrder', 		bNameEditable := FALSE, 		nGS1_AI := 91);
	stCryptoCode					:	ST_CodeValidation	:=		(sFieldName :='CryptoCode', 			bNameEditable := FALSE, 		nGS1_AI := 93);
	stRSKU						:	ST_CodeValidation	:=		(sFieldName :='RSKU', 						bNameEditable := FALSE, 		nGS1_AI := 240);
	stMRP		 				:	ST_CodeValidation	:=		(sFieldName :='MRP', 						bNameEditable := FALSE, 		nGS1_AI := 8005);
	stBrandSpecification			:	ST_CodeValidation	:=		(sFieldName :='BrandSpec',			bNameEditable := FALSE, 		nGS1_AI := 92);
	stProduceDate					:	ST_CodeValidation	:=		(sFieldName :='ProduceDate',			bNameEditable := TRUE, 		nGS1_AI := 94);
	stUserField3					:	ST_CodeValidation	:=		(sFieldName :='',						bNameEditable := TRUE, 		nGS1_AI := 95);

END_STRUCT
END_TYPE

// ---- DUTs/METS/AI Codes And Validation/ST_CodeValidation.TcDUT
TYPE ST_CodeValidation :
STRUCT
	bValidate 			:	BOOL;

	sFieldName		:	STRING(15)	:='';
	bNameEditable	:	BOOL;
	nListPosition		: 	BYTE;

	sStartAI 			: 	STRING(6)		:= '';
	sEndAI 			: 	STRING(6) 	:= '';
	nCodeStartPos		:	INT;
	nCodeLength		:	INT;

	nGS1_AI			: 	INT;

(* If sStartAI is empty, then use nCodeStartPos, else find sStartAI in code for start position *)
(* If sEndAI is empty then use nCodeLength, else find sEndAI in code for end position*)

(*General Application Idendifiers (AI) Description:
	01:		GTIN
	10: 		Batch ID
	21: 		Serial Code
	91:		Production Order
	93:		Crypto
	240:		RSKU
*)

END_STRUCT
END_TYPE

// ---- DUTs/METS/AI Codes And Validation/ST_RejectItems.TcDUT
TYPE ST_RejectItems :
STRUCT
	nRejectID			: UINT;
	sMetsDisplayCode	: T_RejectCode; (*this is what is displayed on our HMI - nn is replaced by the number of failures/successes*)
	sMetsSearchCode		: STRING(50); (*this is what to search for when changing the reject reason for FSS*)
	sFssSendCode		: T_FSS_RejecCode; (*this is what to send to FSS*)
END_STRUCT
END_TYPE

// ---- DUTs/METS/AI Codes And Validation/ST_RejectReasonsForCase.TcDUT
TYPE ST_RejectReasonsForCase :
STRUCT
	stValError:				ST_RejectItems :=(		nRejectID := 301,
														sMetsDisplayCode:='XXVALnnXX',
														sMetsSearchCode:='VAL',
														sFssSendCode:='Validation_DeferredOuter');

	stOACError:				ST_RejectItems :=(	nRejectID := 302,
														sMetsDisplayCode:='XXOACnnXX',
														sMetsSearchCode:='OAC',
														sFssSendCode:='Validation_DeferredPackData');

	stINVError:				ST_RejectItems :=(	nRejectID := 303,
														sMetsDisplayCode:='XXINVnnXX',
														sMetsSearchCode:='INV',
														sFssSendCode:='Validation_BelowAcceptanceLevel');

	stDUPError:				ST_RejectItems :=(	nRejectID := 304,
														sMetsDisplayCode:='XXDUPn1-n2XX',
														sMetsSearchCode:='DUP',
														sFssSendCode:='Validation_DuplicateData');

	stPackNotLinedError:		ST_RejectItems :=(	nRejectID := 305,
														sMetsDisplayCode:='XXPACKnnXX',
														sMetsSearchCode:='XPACK',
														sFssSendCode:='Validation_BadPackCode');

	stOuterGTINError:		ST_RejectItems :=(		nRejectID := 306,
														sMetsDisplayCode:='XXOUTERGTINnnXX',
														sMetsSearchCode:='OUTERGTIN',
														sFssSendCode:='Validation_BadOuterCode');

	stOuterSerialError:		ST_RejectItems :=(		nRejectID := 307,
														sMetsDisplayCode:='XXOUTERSERnnXX',
														sMetsSearchCode:='OUTERSER',
														sFssSendCode:='Validation_BadOuterCode');

	stOuterRSKUError:		ST_RejectItems :=(		nRejectID := 308,
														sMetsDisplayCode:='XXOUTERSKUnnXX',
														sMetsSearchCode:='OUTERSKU',
														sFssSendCode:='Validation_BadOuterCode');

	stNoCaseLabelError:		ST_RejectItems :=(		nRejectID := 309,
														sMetsDisplayCode:='XXNOCASELABELXX',
														sMetsSearchCode:='NOCASELABEL',
														sFssSendCode:='NoReadCase');

	stCasePackerReject:		ST_RejectItems :=(		nRejectID := 310,
														sMetsDisplayCode:='XXCASEPACKERREJECTXX',
														sMetsSearchCode:='CASEPACKERREJECT',
														sFssSendCode:='CasePackerReject');

	stDoorGuardReject:		ST_RejectItems :=(		nRejectID := 311,
														sMetsDisplayCode:='XXDOORGUARDREJECTXX',
														sMetsSearchCode:='DOORGUARDREJECT',
														sFssSendCode:='DoorReject');

	stCaseLabelGtinError:	ST_RejectItems :=(		nRejectID := 312,
														sMetsDisplayCode:='XXCASEGTINXX',
														sMetsSearchCode:='CASEGTIN',
														sFssSendCode:='Validation_BadLabel');

	stCaseLabelRskuError:	ST_RejectItems :=(		nRejectID := 313,
														sMetsDisplayCode:='XXCASESKUXX',
														sMetsSearchCode:='CASESKU',
														sFssSendCode:='Validation_BadLabel');

	stCaseLabelProductionOrderError:	ST_RejectItems :=(	nRejectID := 314,
														sMetsDisplayCode:='XXCASEPRODXX',
														sMetsSearchCode:='CASEPROD',
														sFssSendCode:='Validation_BadLabel');

	stCaseLabelBatchIDError:	ST_RejectItems :=(		nRejectID := 315,
														sMetsDisplayCode:='XXCASEBATCHXX',
														sMetsSearchCode:='CASEBATCH',
														sFssSendCode:='Validation_BadLabel');

	stCaseLabelSerialCodeError:	ST_RejectItems :=(	nRejectID := 316,
														sMetsDisplayCode:='XXCASESERIALCODEXX',
														sMetsSearchCode:='CASESERIALCODE',
														sFssSendCode:='Validation_BadLabel');

	stCaseLabelDuplicate:	ST_RejectItems :=(		nRejectID := 317,
														sMetsDisplayCode:='XXDUPCASELABELXX',
														sMetsSearchCode:='DUPCASELABEL',
														sFssSendCode:='Validation_CaseDuplicate');

	stCaseNoCaseData:	ST_RejectItems :=(			nRejectID := 318,
														sMetsDisplayCode:='XXNOCASEDATAXX',
														sMetsSearchCode:='NOCASEDATA',
														sFssSendCode:='Integrity_TooFewItemsCase');

	stCaseBarcodeInvalidLength:	ST_RejectItems :=(	nRejectID := 319,
														sMetsDisplayCode:='XXCASECODELENGTHXX',
														sMetsSearchCode:='CASECODELENGTH',
														sFssSendCode:='Validation_BadLabel');

	stCaseDBInvalidCheck	:	ST_RejectItems :=(	nRejectID := 320,
														sMetsDisplayCode:='XXCACDBINVALIDXX',
														sMetsSearchCode:='CACDBINVALID',
														sFssSendCode:='Validation_DBInvalid');

	stCaseWhitelistInvalidCheck	:	ST_RejectItems :=(	nRejectID := 321,
														sMetsDisplayCode:='XXOHMWHITELISTXX',
														sMetsSearchCode:='OHMWHITELIST',
														sFssSendCode:='Validation_OHMWhitelistInvalid');

	stOuterBrandError				:	ST_RejectItems :=(	nRejectID := 322,
														sMetsDisplayCode:='XXOUTERSBRANDnnXX',
														sMetsSearchCode:='OUTERSBRAND',
														sFssSendCode:='Validation_BadOuterCode');

	stCaseLabelBrandCodeError:	ST_RejectItems :=(	nRejectID := 323,
														sMetsDisplayCode:='XXCASEBRANDXX',
														sMetsSearchCode:='CASEBRAND',
														sFssSendCode:='Validation_BadLabel');

	stUnknownCaseReject:		ST_RejectItems :=(	nRejectID := 300,
														sMetsDisplayCode:='UnknownReason',
														sMetsSearchCode:='UnknownReason',
														sFssSendCode:='UnknownReason');

END_STRUCT
END_TYPE

// ---- DUTs/METS/AI Codes And Validation/ST_RejectReasonsForOuter.TcDUT
TYPE ST_RejectReasonsForOuter :
STRUCT
	stOuterBarcodeGtinError:		ST_RejectItems :=(	nRejectID := 201,
															sMetsDisplayCode:='Outer code invalid GTIN',
															sMetsSearchCode:='GTIN',
															sFssSendCode:='WrongMasterData');

	stOuterBarcodeRskuError:	ST_RejectItems :=(	nRejectID := 202,
															sMetsDisplayCode:='Outer code invalid RSKU',
															sMetsSearchCode:='RSKU',
															sFssSendCode:='WrongMasterData');

	stOuterCodeSerialError:		ST_RejectItems :=(	nRejectID := 203,
															sMetsDisplayCode:='Outer code invalid lenght Serial Code',
															sMetsSearchCode:='Serial',
															sFssSendCode:='Validation_BadCode');

	stOuterBarcodeInvalidLength:	ST_RejectItems :=(	nRejectID := 204,
															sMetsDisplayCode:='Outer code invalid Length',
															sMetsSearchCode:='Length',
															sFssSendCode:='Validation_BadCode');

	stOuterBarcodeNotRead:		ST_RejectItems :=(	nRejectID := 205,
															sMetsDisplayCode:='Outer Label Code Not Read',
															sMetsSearchCode:='Outer Label Code Not Read',
															sFssSendCode:='NoReadOuter');

	stOuterBarcodeDuplicate:	ST_RejectItems :=(	nRejectID := 206,
															sMetsDisplayCode:='Outer code duplicate',
															sMetsSearchCode:='code duplicate',
															sFssSendCode:='Validation_OuterDup');

	stOuterDataNotFound:		ST_RejectItems :=(	nRejectID := 207,
															sMetsDisplayCode:='Outer data (OAC) not found',
															sMetsSearchCode:='(OAC) not found',
															sFssSendCode:='NoReadOuterData');

	stOuterGeneralCodeError:	ST_RejectItems :=(	nRejectID := 208,
															sMetsDisplayCode:='No Codes Read At Aggregation Station',
															sMetsSearchCode:='No Codes Read At Aggregation Station',
															sFssSendCode:='Validation_General');

	stOuterTimeOutValidation:	ST_RejectItems :=(	nRejectID := 209,
															sMetsDisplayCode:='Outer Validation Timeout',
															sMetsSearchCode:='Validation Timeout',
															sFssSendCode:='Validation_General');

(*Outer general erros related to pack codes only - barcode validation - OK*)

	stOuterDuplicatedPackCodesFound:		ST_RejectItems :=(	nRejectID := 210,
															sMetsDisplayCode:='Outer contain duplicate pack codes',
															sMetsSearchCode:='duplicate pack codes',
															sFssSendCode:='Validation_PackDup');

	stOuterPackCodeDataNotFound:		ST_RejectItems :=(	nRejectID := 211,
															sMetsDisplayCode:='Outer - Pack codes data (OCV) not found',
															sMetsSearchCode:='OCV',
															sFssSendCode:='NoPacksCodeData');

	stOuterConfirmCodeNotRead:			ST_RejectItems :=(	nRejectID := 212,
															sMetsDisplayCode:= 'Interim code(s) not read',
															sMetsSearchCode:='Interim code(s) not read',
															sFssSendCode:='NoPackCodeData');

	stOuterPackCodeNotRead:				ST_RejectItems :=(	nRejectID := 213,
															sMetsDisplayCode:= 'Outer acceptance level - n1 of n2 pack codes read',
															sMetsSearchCode:='acceptance level',
															sFssSendCode:='Tolerance_PackNoRead');

	stOuterPackCodeInvalid:				ST_RejectItems :=(	nRejectID := 214,
															sMetsDisplayCode:= 'Outer - invalid pack code(s) found',
															sMetsSearchCode:='Outer - invalid pack',
															sFssSendCode:='Tolerance_PackInv');

(*Outer external rejeqt for quality - barcode validation - OK, pack codes(s) validation - OK*)

	stOuterQAReject:			ST_RejectItems :=(	nRejectID := 215,
															sMetsDisplayCode:='Outer QA Reject',
															sMetsSearchCode:='QA',
															sFssSendCode:='QA_Reject');

	stOuterPackCodeDBError:				ST_RejectItems :=(	nRejectID := 216,
															sMetsDisplayCode:= 'Number Pack code not found - n1 of n2 - DB Error',
															sMetsSearchCode:='pack codes DB Error',
															sFssSendCode:='Validation_BadDB');

	stOuterBarcodeDBError:				ST_RejectItems :=(	nRejectID := 217,
															sMetsDisplayCode:= 'Outer code not found  - DB Error',
															sMetsSearchCode:='Outer code DB Error',
															sFssSendCode:='Validation_BadDB');

	stOuterCodesBrandSpecError	:		ST_RejectItems :=(	nRejectID := 218,
														sMetsDisplayCode:='Outer code invalid Brand',
														sMetsSearchCode:='Outer code invalid Brand',
														sFssSendCode:='Validation_BadCode');


	stUnknownOuterReject:		ST_RejectItems :=(	nRejectID := 200,
															sMetsDisplayCode:='',
															sMetsSearchCode:='',
															sFssSendCode:='UnknownReason');

END_STRUCT
END_TYPE

// ---- DUTs/METS/AI Codes And Validation/ST_RejectReasonsForPack.TcDUT
TYPE ST_RejectReasonsForPack :
STRUCT
	stPackCodesNotLinked:		ST_RejectItems :=(	nRejectID := 101,
														sMetsDisplayCode:='Pack code(s) not linked',
														sMetsSearchCode:='Pack code(s) not linked',
														sFssSendCode:='NoPackData');

	stPackCodesOverwritten:		ST_RejectItems :=(	nRejectID := 102,
														sMetsDisplayCode:='Pack code(s) over-written',
														sMetsSearchCode:='Pack code(s) over-written',
														sFssSendCode:='WrongReadPackCode');

	stPackCodesGtinError:		ST_RejectItems :=(	nRejectID := 103,
														sMetsDisplayCode:='Pack code(s) invalid GTIN',
														sMetsSearchCode:='Pack code(s) invalid GTIN',
														sFssSendCode:='WrongMasterData');

	stPackCodesSerialError:		ST_RejectItems :=(	nRejectID := 104,
														sMetsDisplayCode:='Pack code(s) invalid Serial Code',
														sMetsSearchCode:='Pack code(s) invalid Serial Code',
														sFssSendCode:='Validation_BadCode');

	stPackCodeInvalidLength	:	ST_RejectItems :=(	nRejectID := 105,
														sMetsDisplayCode:='Pack code(s) invalid Length',
														sMetsSearchCode:='Pack code(s) invalid Length',
														sFssSendCode:='Validation_BadCode');

	stPackCodesNotRead:		ST_RejectItems :=(	nRejectID := 106,
														sMetsDisplayCode:='Pack code(s) no read',
														sMetsSearchCode:='Pack code(s) no read',
														sFssSendCode:='NoReadPackCode');

	stPackCodesDuplicated:		ST_RejectItems :=(	nRejectID := 107,
														sMetsDisplayCode:='Pack code(s) duplicate',
														sMetsSearchCode:='Pack code(s) duplicate',
														sFssSendCode:='Validation_BadCode');

	stPackCodesTypeError:		ST_RejectItems :=(	nRejectID := 108,
														sMetsDisplayCode:='Pack code(s) invalid type',
														sMetsSearchCode:='Pack code(s) invalid type',
														sFssSendCode:='Validation_BadType');

	stPackCodesSUPIError:		ST_RejectItems :=(	nRejectID := 109,
														sMetsDisplayCode:='Pack code(s) SUPI failed validation',
														sMetsSearchCode:='Pack code(s) SUPI failed validation',
														sFssSendCode:='Validation_BadSUPI');


	stPackCodesDBError:		ST_RejectItems :=(	nRejectID := 110,
														sMetsDisplayCode:='Pack code DB failed validation',
														sMetsSearchCode:='Pack code DB failed validation',
														sFssSendCode:='Validation_BadDB');

	stPackCodesBrandSpec:		ST_RejectItems :=(	nRejectID := 111,
														sMetsDisplayCode:='Pack code(s) invalid Brand',
														sMetsSearchCode:='Pack code(s) invalid Brand',
														sFssSendCode:='Validation_BadCode');


	stUnknownPackReject:		ST_RejectItems :=(	nRejectID := 100,
														sMetsDisplayCode:='UnknownReason',
														sMetsSearchCode:='UnknownReason',
														sFssSendCode:='UnknownReason');


END_STRUCT
END_TYPE

// ---- DUTs/METS/Alarms/E_MessageType.TcDUT
{attribute 'qualified_only'}
//{attribute 'strict'}
//{attribute 'to_string'}
TYPE E_MessageType :
(
	DISABLEBYMESSAGETYPE		:=-1,
	GENERALSYSTEMALARM 		:=0,				(*Message type 0*)
	EUCASUBSYSTEMALARM 		:=1,				(*Message type 1*)
	TPDSUBSYSTEMALARM 		:=2,				(*Message type 2*)
	EXTERNALALARM 			:=3,				(*Message type 3*)
	SPARE04ALARM				:=4,				(*Message type 4*)
	SPARE05ALARM	 			:=5,				(*Message type 5*)
	SPARE06ALARM	 			:=6,				(*Message type 6*)
	SPARE07ALARM				:=7,				(*Message type 7*)


	GENERALSYSTEMWARNING 	:=8,				(*Message type 8*)
	EUCASUBSYSTEMWARNING 	:=9,				(*Message type 9*)
	TPDSUBSYSTEMWARNING 	:=10,				(*Message type 10*)
	EXTERNALWARNING 			:=11,				(*Message type 11*)
	SPARE12WARNING 			:=12,				(*Message type 12*)
	SPARE13WARNING 			:=13,				(*Message type 13*)
	SPARE14WARNING 			:=14,				(*Message type 14*)
	SPARE15WARNING 			:=15				(*Message type 15*)

);
END_TYPE

// ---- DUTs/METS/Alarms/ST_AlarmDB.TcDUT
TYPE ST_AlarmDB :
STRUCT
	eEventID			: E_MessageID;
	eRootEventID		: E_MessageID;
	nEventCat			: INT;
	nEventTypeNo		: INT;
	sEventTypeID		: STRING(1);
	sEquipmentName		: STRING;
	bIsActive			: BOOL;
	sEventStart			: STRING;
	sEventEnd			: STRING;
END_STRUCT
END_TYPE

// ---- DUTs/METS/Alarms/ST_Alarms.TcDUT
TYPE ST_Alarms :
STRUCT
	nMessage						: 	DWORD;
	nMessageTimer				:	ARRAY[0..31] OF TON;
	nCategory						:	ARRAY[0..31] OF INT;
	nMessageType					:	WORD;
END_STRUCT
END_TYPE

// ---- DUTs/METS/Alarms/ST_AlarmSettings.TcDUT
TYPE ST_AlarmSettings :
STRUCT
	aTextMessageTable		: ARRAY [0..31] OF STRING(200);
	aAlarmTriggerTable		: ARRAY [0..31] OF BOOL;

	aAlarmTimoutTable		: ARRAY [0..31] OF TIME;
	aBlockEnableTable			: ARRAY [0..31] OF BOOL :=[ 32 (FALSE)];
	aInhibitResetTable			: ARRAY [0..31] OF BOOL;
	aAutoResetTable			: ARRAY[0..31] OF BOOL;
	aInternalResetTable		: ARRAY [0..31] OF BOOL;

	aCategoryNoTable			: ARRAY[0..31] OF INT;
	aMessageTypeStatusTable	: ARRAY[0..31] OF WORD;
END_STRUCT
END_TYPE

// ---- DUTs/METS/Alarms/ST_AlarmsTable.TcDUT
TYPE ST_AlarmsTable :
STRUCT
	aTextMessages	 					: 	ARRAY [0..cMAX_MESSAGE_NUMBER] OF STRING(200);
	aActiveID							: 	ARRAY [0..cMAX_MESSAGE_NUMBER] OF BOOL;
	aDisableAlarmLog					:	ARRAY [0..cMAX_MESSAGE_NUMBER] OF BOOL;


	aMsgHMI							:	ARRAY [0..cMAX_MESSAGE_NUMBER] OF T_MaxString;
	aAlarmDB							:	ARRAY [0..cMAX_MESSAGE_NUMBER] OF ST_AlarmDB;
	aMsgAux							:	ARRAY [0..cMAX_MESSAGE_NUMBER] OF ST_ALARM_Aux;
	
	
	aLogMessages						:	ARRAY[1..cMAX_DISPLAY_ALARMS] OF STRING(200);
	aActiveMessages					:	ARRAY[1..15] OF STRING(200);
	aActiveMessagesHMI				:	ARRAY[1..15] OF INT:=[ 15(-1)];

	aLogAlarmsHMI						:	ARRAY[1..cMAX_DISPLAY_ALARMS] OF INT :=[ cMAX_DISPLAY_ALARMS(-1)];
	aLogWarningsHMI					:	ARRAY[1..cMAX_DISPLAY_ALARMS] OF INT :=[ cMAX_DISPLAY_ALARMS(-1)];
	aLogDateAlarmsHMI					:	ARRAY[1..cMAX_DISPLAY_ALARMS] OF STRING(19);	(* date/time as HH:MM:SS DD/MM/YYYY for HMI display *)
	aLogDateWarningsHMI				:	ARRAY[1..cMAX_DISPLAY_ALARMS] OF STRING(19);	(* date/time as HH:MM:SS DD/MM/YYYY for HMI display *)
END_STRUCT
END_TYPE

// ---- DUTs/METS/Alarms/ST_AlarmStatus.TcDUT
TYPE ST_AlarmStatus :
STRUCT
	bNoActiveAlarms					: BOOL;
	bNoActiveWarrnings				: BOOL;

	bGeneralSystemAlarmActive		: BOOL;		(*Message type 0*)
	bEUCASubsytemAlarmActive		: BOOL;		(*Message type 1*)
	bTPDSubsytemAlarmActive		: BOOL;		(*Message type 2*)
	bExternalAlarmActive				: BOOL;		(*Message type 3*)

	bSpare04AlarmActive				: BOOL;		(*Message type 4*)
	bSpare05AlarmActive				: BOOL;		(*Message type 5*)
	bSpare06AlarmActive				: BOOL;		(*Message type 6*)
	bSpare07AlarmActive				: BOOL;		(*Message type 7*)

	bGeneralSystemWarningActive		: BOOL;		(*Message type 8*)
	bEUCASubsytemWarningActive	: BOOL;		(*Message type 9*)
	bTPDSubsytemWarningActive		: BOOL;		(*Message type 10*)
	bExternalWarningActive			: BOOL;		(*Message type 11*)

	bSpare12WarningActive			: BOOL;		(*Message type 12*)
	bSpare13WarningActive			: BOOL;		(*Message type 13*)
	bSpare14WarningActive			: BOOL;		(*Message type 14*)
	bSpare15WarningActive			: BOOL;		(*Message type 15*)

	(*eMessageType					: E_MessageType;*)
END_STRUCT
END_TYPE

// ---- DUTs/METS/Aliases/T_CAC_Filename.TcDUT
TYPE T_CAC_Filename : T_MaxString;
END_TYPE

// ---- DUTs/METS/Aliases/T_CASE_Barcode.TcDUT
TYPE T_CASE_Barcode : T_MaxString;
END_TYPE

// ---- DUTs/METS/Aliases/T_Char.TcDUT
TYPE T_Char : STRING[1];
END_TYPE

// ---- DUTs/METS/Aliases/T_CHM_Filename.TcDUT
TYPE T_CHM_Filename : T_MaxString;
END_TYPE

// ---- DUTs/METS/Aliases/T_CodeBATCH.TcDUT
 TYPE T_CodeBATCH : STRING[10];
END_TYPE

// ---- DUTs/METS/Aliases/T_CodeBRAND.TcDUT
 TYPE T_CodeBRAND : STRING[9];
END_TYPE

// ---- DUTs/METS/Aliases/T_CodeCRYPTO.TcDUT
TYPE T_CodeCRYPTO : STRING[20];
END_TYPE

// ---- DUTs/METS/Aliases/T_CodeGTIN.TcDUT
TYPE T_CodeGTIN : STRING[20];
END_TYPE

// ---- DUTs/METS/Aliases/T_CodeMRP.TcDUT
TYPE T_CodeMRP : STRING[8];
END_TYPE

// ---- DUTs/METS/Aliases/T_CodePIT.TcDUT
TYPE T_CodePIT : STRING[7];
END_TYPE

// ---- DUTs/METS/Aliases/T_CodePO.TcDUT
TYPE T_CodePO : STRING[20];
END_TYPE

// ---- DUTs/METS/Aliases/T_CodePRODUCEDATE.TcDUT
 TYPE T_CodePRODUCEDATE : STRING[14];
END_TYPE

// ---- DUTs/METS/Aliases/T_CodeRSKU.TcDUT
 TYPE T_CodeRSKU : STRING[9];
END_TYPE

// ---- DUTs/METS/Aliases/T_CodeURL.TcDUT
TYPE T_CodeURL : STRING[20];
END_TYPE

// ---- DUTs/METS/Aliases/T_DB_LongSTRING.TcDUT
TYPE T_DB_LongSTRING : STRING(1024);
END_TYPE

// ---- DUTs/METS/Aliases/T_FileExtension.TcDUT
TYPE T_FileExtension : STRING[4];
END_TYPE

// ---- DUTs/METS/Aliases/T_FolderName.TcDUT
TYPE T_FolderName : STRING[25];
END_TYPE

// ---- DUTs/METS/Aliases/T_FolderPath.TcDUT
TYPE T_FolderPath : STRING[100];
END_TYPE

// ---- DUTs/METS/Aliases/T_FSS_RejecCode.TcDUT
TYPE T_FSS_RejecCode : STRING(40);
END_TYPE

// ---- DUTs/METS/Aliases/T_HMI_PACK_Barcode.TcDUT
TYPE T_HMI_PACK_Barcode : STRING(cMAX_HMI_PACKCODE_LENGHT);
END_TYPE

// ---- DUTs/METS/Aliases/T_ISO8601Time.TcDUT
TYPE T_ISO8601Time : STRING(30);
END_TYPE

// ---- DUTs/METS/Aliases/T_LongSTRING.TcDUT
TYPE T_LongSTRING : STRING(1023);
END_TYPE

// ---- DUTs/METS/Aliases/T_OAC_Filename.TcDUT
TYPE T_OAC_Filename : T_MaxString;
END_TYPE

// ---- DUTs/METS/Aliases/T_OCV_Filename.TcDUT
TYPE T_OCV_Filename : T_MaxString;
END_TYPE

// ---- DUTs/METS/Aliases/T_OHM_Filename.TcDUT
TYPE T_OHM_Filename : STRING(44);
END_TYPE

// ---- DUTs/METS/Aliases/T_OUTER_Barcode.TcDUT
TYPE T_OUTER_Barcode : T_MaxString;
END_TYPE

// ---- DUTs/METS/Aliases/T_PACK_Barcode.TcDUT
TYPE T_PACK_Barcode : STRING(cMAX_PACKCODE_LENGHT);
END_TYPE

// ---- DUTs/METS/Aliases/T_PCM_Filename.TcDUT
 TYPE T_PCM_Filename : T_MaxString;
END_TYPE

// ---- DUTs/METS/Aliases/T_PositiveDINT.TcDUT
TYPE T_PositiveDINT : DINT(0..2147483647); END_TYPE

// ---- DUTs/METS/Aliases/T_PositiveINT.TcDUT
TYPE T_PositiveINT : INT(0..32767); END_TYPE

// ---- DUTs/METS/Aliases/T_ProductDescription.TcDUT
TYPE T_ProductDescription : STRING[48];
END_TYPE

// ---- DUTs/METS/Aliases/T_RejectCode.TcDUT
TYPE T_RejectCode : STRING[100];
END_TYPE

// ---- DUTs/METS/Aliases/T_TimeLog.TcDUT
TYPE T_TimeLog : STRING[15];
END_TYPE

// ---- DUTs/METS/Case/CAC/E_CAC_State.TcDUT
TYPE E_CAC_State :
(
	E_CAC_IDLE,
	E_CAC_OPENFILE,
	E_CAC_BUILDXMLIMAGE,
	E_CAC_WRITEXMLIMAGE,
	E_CAC_CLOSEXMLIMAGE,
	E_CAC_CLOSEFILE,
	E_CAC_FINDFOLDER,
	E_CAC_FINDFILE,
	E_CAC_READDATA,
	E_CAC_WRITEDATA,
	E_CAC_CREATEFOLDER,
	E_CAC_DELETEFOLDER,
	E_CAC_DELETEFILE,
	E_CAC_CREATEOACDATA,
	E_CAC_CREATEOCVDATA,
	E_CAC_WRITEOCVDATA,
	E_CAC_DELETEOAC,
	E_CAC_DELETEOCV1,
	E_CAC_DELETEOCV2,
	E_CAC_COPYFILE,
	E_CAC_MOVEFILE,
	E_CAC_RENAMEFILE,
	E_CAC_VALIDATECASE 			:= 22,
	E_CAC_VALIDATEOUTER,
	E_CAC_VALIDATEOAC,
	E_CAC_VALIDATEPACK,
	E_CAC_DUPLICATEOUTERCHECK,
	E_CAC_DBREQUEST,
	E_CAC_DBRESPONSE,
	E_CAC_CHECKOUTERDUPLICATES,
	E_CAC_CHECKPACKDUPLICATES,
	E_CAC_DONE					:= 31
);
END_TYPE

// ---- DUTs/METS/Case/CAC/ST_CAC_Data.TcDUT
TYPE ST_CAC_Data :
STRUCT
	Barcode 				: T_CASE_Barcode;
	ProductionDate			: STRING(10);
	ProductionTime			: STRING(8);
	ProductionTimeOffset	: STRING(6);		(* time offset between system and UTC, '+1:00' means SystemTime = UTC + 1hr *)
	RetailSKU				: T_CodeRSKU;
	CasePacker				: ST_SYSTEM_MachineID;
	CodingAndTrackingMode	: INT;
	NumberOfOuters			: INT;
	CaseRejectCode			: T_RejectCode; (* blank and not included in CAC files for valid cases *)
	CaseRejectID			: UINT	; (* blank and not included in CAC files for valid cases *)
	Outer					: ARRAY[1..cMAX_OUTERS_PER_CASE] OF ST_OAC_Data;
END_STRUCT
END_TYPE

// ---- DUTs/METS/Case/CHM/CHM Data Structure/GenericHierarchy/Case Item Structures/ST_CaseContent.TcDUT
TYPE ST_CaseContent :
STRUCT
	DefaultIdentity 		: ST_DefaultIdentity;
	ExpectedItemCount	: STRING(3);
	ItemReadRate			: STRING(3);
	arrOuterItem			: ARRAY[1..cMAX_OUTERS_PER_CASE] OF ST_OuterItem;

END_STRUCT
END_TYPE

// ---- DUTs/METS/Case/CHM/CHM Data Structure/GenericHierarchy/Case Item Structures/ST_CaseIdentity.TcDUT
TYPE ST_CaseIdentity :
STRUCT
		SKU			: T_CodeRSKU;
		GTIN			: T_CodeGTIN;
		ID			:STRING(cMAX_CHM_CASEID_LENGHT);
		URL		:T_CodeURL;
		ReadQuality	:STRING(6);

END_STRUCT
END_TYPE

// ---- DUTs/METS/Case/CHM/CHM Data Structure/GenericHierarchy/Case Item Structures/ST_CaseItem.TcDUT
TYPE ST_CaseItem :
STRUCT
	Identity				: 	ST_CaseIdentity;
	ItemState				:	STRING(15);
	RejectReason			: T_FSS_RejecCode;
	TimeStamp				: T_ISO8601Time;
	NoRead				:	STRING(5);
	Content				:	ST_CaseContent;
	ProductionOrder		:	T_CodePO;
	LocalProductionOrder	: T_CodePO;
	PITCode				:	T_CodePIT;
	BatchID				:	T_CodeBATCH;
	ProductionLine			:	STRING(4);
END_STRUCT
END_TYPE

// ---- DUTs/METS/Case/CHM/CHM Data Structure/GenericHierarchy/Outer Item Structures/ST_OuterContent.TcDUT
TYPE ST_OuterContent :
STRUCT
	DefaultIdentity 	: ST_DefaultIdentity;
	ExpectedItemCount		:STRING(3);
	ItemReadRate			:STRING(3);
	arrPackItem			:ARRAY[1..cMAX_PACKS_PER_OUTER] OF ST_PackItem;

END_STRUCT
END_TYPE

// ---- DUTs/METS/Case/CHM/CHM Data Structure/GenericHierarchy/Outer Item Structures/ST_OuterIdentity.TcDUT
TYPE ST_OuterIdentity :
STRUCT

		ID			:STRING(cMAX_CHM_OUTERID_LENGHT);
		URL		:T_CodeURL;
		ReadQuality	:STRING(6);

END_STRUCT
END_TYPE

// ---- DUTs/METS/Case/CHM/CHM Data Structure/GenericHierarchy/Outer Item Structures/ST_OuterItem.TcDUT
TYPE ST_OuterItem :
STRUCT
	Identity				: 	ST_OuterIdentity;
	ItemState				:	STRING(15);
	RejectReason			: T_FSS_RejecCode;
	TimeStamp				: T_ISO8601Time;
	NoRead				:	STRING(5);
	Content				:	ST_OuterContent;

END_STRUCT
END_TYPE

// ---- DUTs/METS/Case/CHM/CHM Data Structure/GenericHierarchy/Pack Item Structures/ST_PackIdentity.TcDUT
TYPE ST_PackIdentity :
STRUCT

		ID			:STRING(cMAX_CHM_PACKID_LENGHT);
		URL		:T_CodeURL;
		ReadQuality	:STRING(6);

END_STRUCT
END_TYPE

// ---- DUTs/METS/Case/CHM/CHM Data Structure/GenericHierarchy/Pack Item Structures/ST_PackItem.TcDUT
TYPE ST_PackItem :
STRUCT
	Identity				: 	ST_PackIdentity;
	ItemState				:	STRING(15);
	RejectReason			: T_FSS_RejecCode;
	TimeStamp				: T_ISO8601Time;
	NoRead				:	STRING(5);

END_STRUCT
END_TYPE

// ---- DUTs/METS/Case/CHM/CHM Data Structure/GenericHierarchy/ST_DefaultIdentity.TcDUT
TYPE ST_DefaultIdentity :
STRUCT

		SKU						: T_CodeRSKU;
		GTIN						: T_CodeGTIN;
		ProductionOrder			: T_CodePO;
		LocalProductionOrder		: T_CodePO;
		PITCode					:T_CodePIT;
		BatchID					:T_CodeBATCH;
		ProductionLine				:STRING(4);

END_STRUCT
END_TYPE

// ---- DUTs/METS/Case/CHM/CHM Data Structure/ST_Attributes.TcDUT
TYPE ST_Attributes :
STRUCT

	ProduceDateMC			: STRING(14);

END_STRUCT
END_TYPE

// ---- DUTs/METS/Case/CHM/CHM Data Structure/ST_CHM_GenericHierarchy.TcDUT
TYPE ST_CHM_GenericHierarchy :
STRUCT
	HierarchyType		:	STRING(5);
	PerformedAction	:	STRING(10);
	TrackingLevels		:	STRING(10);
	TrackingIndicator	:	STRING(3);
	CaseItem			:	ST_CaseItem;

END_STRUCT
END_TYPE

// ---- DUTs/METS/Case/CHM/CHM Data Structure/ST_GenericHierarchy.TcDUT
TYPE ST_GenericHierarchy :
STRUCT
	HierarchyType		:	STRING(5);
	PerformedAction	:	STRING(10);
	TrackingLevels		:	STRING(10);
	TrackingIndicator	:	STRING(3);
	CaseItem			:	ST_CaseItem;

END_STRUCT
END_TYPE

// ---- DUTs/METS/Case/CHM/CHM Data Structure/ST_MessageHeader.TcDUT
TYPE ST_MessageHeader :
STRUCT

	(*CreationDate 				: STRING(10);
	CreationTime 				: STRING(25);*)
	ReferenceID				: T_MaxString;
	CreationTimeLocalUTC		: T_ISO8601Time;
	MessageType	 			: STRING(25);
	SenderSystem				: STRING(5);
	ReceiverSystem			: STRING(5);


END_STRUCT
END_TYPE

// ---- DUTs/METS/Case/CHM/E_CHM_GeneratorState.TcDUT
TYPE E_CHM_GeneratorState :
(
	E_CHM_IDLEGENERATOR,
	E_CHM_FILECHECK,
	E_CHM_FILEOPEN,
	E_CHM_GENERATEHEAD,
	(*E_CHM_HEADDONE,*)
	E_CHM_GENERATEBODY,
	(*E_CHM_BODYDONE,*)
	E_CHM_GENERATEENDING,
	(*E_CHM_ENDINGDONE,*)
	E_CHM_FILECLOSE,
	E_CHM_GENERATEFLG,
	(*E_CHM_FLGDONE,*)
	E_CHM_TIMEOUT,
	E_CHM_DONEGENERATOR
);
END_TYPE

// ---- DUTs/METS/Case/CHM/E_CHM_State.TcDUT
TYPE E_CHM_State :
(
	E_CHM_IDLE,
	E_CHM_OPENFILE,
	E_CHM_BUILDXMLIMAGE,
	E_CHM_WRITEXMLIMAGE,
	E_CHM_CLOSEFILE,
	E_CHM_FINDFOLDER,
	E_CHM_FINDFILE,
	E_CHM_READDATA,
	E_CHM_WRITEDATA,
	E_CHM_CREATEFOLDER,
	E_CHM_DELETEFOLDER,
	E_CHM_DELETEFILE,
	E_CHM_COPYFILE,
	E_CHM_MOVEFILE,
	E_CHM_RENAMEFILE,
	E_CHM_VALIDATECASE,
	E_CHM_VALIDATEOUTER,
	E_CHM_VALIDATEOAC,
	E_CHM_VALIDATEPACK,
	E_CHM_DUPLICATEOUTERCHECK,
	E_CHM_DONE
);
END_TYPE

// ---- DUTs/METS/Case/CHM/E_CHM_WriteMode.TcDUT
TYPE E_CHM_WriteMode :
(
	E_CHM_FSS2MODE_NOBACKUP,
	E_CHM_FSS2MODE_FSS2BACKUP,
	E_CHM_FSS3MODE_NOBACKUP,
	E_CHM_FSS3MODE_FSS2BACKUP

);
END_TYPE

// ---- DUTs/METS/Case/CHM/ST_CHM_Data.TcDUT
TYPE ST_CHM_Data :
STRUCT
	MessageHeader		:	ST_MessageHeader;
	Factory				:	STRING(3);
	GenericHierarchy		:	ST_GenericHierarchy;
	Attributes				:	ST_Attributes;
END_STRUCT
END_TYPE

// ---- DUTs/METS/Case/E_CASE_State.TcDUT
TYPE E_CASE_State :
(
	E_CASE_IDLE,
	E_CASE_SCANINFEEDQUEUE,
	E_CASE_COPYOACFILE,
	E_CASE_READOACDATA,
	E_CASE_SCANOUTERS,
	E_CASE_DUPLICATEPACKCHECK,
	E_CASE_UPDATEINFEEDQUEUE,
	E_CASE_DELETEOACFILE,
	E_CASE_DELETEOCV1FILE,
	E_CASE_DELETEOCV2FILE,
	E_CASE_VALIDATECAC,
	E_CASE_GETSERIALCODE,
	E_CASE_FINDCACFILE,
	E_CASE_RENAMECACFILE,
	E_CASE_MOVECACFILE,
	E_CASE_DATAVALIDATE,
	E_CASE_DATAWRITEXML,
	E_CASE_OVERWIRTECAC,
	E_CASE_DATAFINALISE,
	E_CASE_DONE
);
END_TYPE

// ---- DUTs/METS/Case/ORCA/E_ORCA_State.TcDUT
TYPE E_ORCA_State :
(
	E_ORCA_IDLE,
	E_ORCA_OPENFILE,

	E_ORCA_CLOSEFILE,
	E_ORCA_FINDFOLDER,
	E_ORCA_FINDFILE,
	E_ORCA_READDATA,

	E_ORCA_DELETEFILE,
	E_ORCA_COPYFILE,
	E_ORCA_MOVEFILE,
	E_ORCA_RENAMEFILE,

	E_ORCA_VALIDATEOUTER,
	E_ORCA_VALIDATEOAC,

	E_ORCA_DONE
);
END_TYPE

// ---- DUTs/METS/Case/ORCA/ST_ORCA_BrandInfo.TcDUT
TYPE ST_ORCA_BrandInfo :
STRUCT

	BatchID 			: STRING(255);
	GTIN 			: STRING(255);
	SKU 				: STRING(255);
	ProductionOrder 	: STRING(255);

END_STRUCT
END_TYPE

// ---- DUTs/METS/Case/ORCA/ST_ORCA_Data.TcDUT
TYPE ST_ORCA_Data :
STRUCT
	SiteInfo 				: ST_ORCA_SiteInfo;
	BrandInfo 			: ST_ORCA_BrandInfo;
	ProductInfo			: ST_ORCA_ProductInfo;
	Outers				: ARRAY[1..60] OF ST_ORCA_Outers;

END_STRUCT
END_TYPE

// ---- DUTs/METS/Case/ORCA/ST_ORCA_Outers.TcDUT
TYPE ST_ORCA_Outers :
STRUCT
	Code 	: STRING(255);
	xPos		: INT;
	yPos		: INT;

END_STRUCT
END_TYPE

// ---- DUTs/METS/Case/ORCA/ST_ORCA_ProductInfo.TcDUT
TYPE ST_ORCA_ProductInfo :
STRUCT

	OutersPerRow 			: STRING(255);
	RowsPerCase	 		: STRING(255);


END_STRUCT
END_TYPE

// ---- DUTs/METS/Case/ORCA/ST_ORCA_SiteInfo.TcDUT
TYPE ST_ORCA_SiteInfo :
STRUCT

	ProductionSite 			: STRING(255);
	ProductionLine 		: STRING(255);


END_STRUCT
END_TYPE

// ---- DUTs/METS/Case/ST_CasePackerInfo.TcDUT
TYPE ST_CasePackerInfo :	(* 8 bytes *)
STRUCT
	ProductionSite 	: STRING(4);
	ProductionLine 	: STRING(4);
END_STRUCT
END_TYPE

// ---- DUTs/METS/Case/ST_CASE_CaseQueue.TcDUT
TYPE ST_CASE_CaseQueue :
STRUCT
	aCACData		: ARRAY[1..cMAX_CASE_QUEUE] OF ST_CAC_Data;	(* array of CAC data *)
	stPrintCACData	: ST_CAC_Data;	(* CAC data sent to printer *)

	stPrintCHMData	: ST_CHM_Data;	(* CHM data printed to XML file *)
END_STRUCT
END_TYPE

// ---- DUTs/METS/Case/ST_CASE_DefferOuter.TcDUT
TYPE ST_CASE_DefferOuter :
STRUCT
	sID 					: STRING(255);
	ProductionDate 		: STRING(10);
	ProductionTime 		: STRING(8);
	ProductionTimeOffset 	: STRING(6);
	RejectCode 			: STRING(255);
END_STRUCT
END_TYPE

// ---- DUTs/METS/Case/ST_CASE_InfeedQueue.TcDUT
TYPE ST_CASE_InfeedQueue :
STRUCT
	nIndex			: T_PositiveINT;				(* number of Outers in queue *)
	sLastBarcode		: T_OUTER_Barcode;	(* last Outer barcode added to Infeed Queue *)
	bDoorReject		: BOOL;
	aOuter			: ARRAY[1..cMAX_INFEED_QUEUE] OF ST_OAC_Data;	(* array of Outer OAC data *)
END_STRUCT
END_TYPE

// ---- DUTs/METS/Device/CX Unit/Device/E_CX_DeviceState.TcDUT
{attribute 'qualified_only'}
{attribute 'strict'}
TYPE E_CX_DeviceState : (
	IDLE,
	ID,
	DEVTYPE,
	BUILDLINES,
	WRITELINE1,
	WRITELINE2,
	ERROR,
	DONE

	//E_CX_DEVICE_CX1,
	//E_CX_DEVICE_CX2
);
END_TYPE

// ---- DUTs/METS/Device/CX Unit/EtherCAT/ST_CX_EtherCATDeviceState.TcDUT
TYPE ST_CX_EtherCATDeviceState :
STRUCT
	bPresent		: BOOL;
	bOpMode			: BOOL;
	bError			: BOOL;
	nDeviceState	: BYTE;
	nLinkState		: BYTE;
	strStatus		: STRING(17);
END_STRUCT
END_TYPE

// ---- DUTs/METS/Device/CX Unit/EtherCAT/ST_CX_EtherCATMasterPNetState.TcDUT
TYPE ST_CX_EtherCATMasterPNetState :
STRUCT
	arrADSAddr		: ARRAY[0..5] OF BYTE;
	nPortNo			: UINT;
	arrAoeAddr		: ARRAY[0..5] OF BYTE;
	nDevState		: UINT;
	nPnIoError		: UINT;
	nPnIoDiag			: UINT;
END_STRUCT
END_TYPE

// ---- DUTs/METS/Device/CX Unit/EtherCAT/ST_CX_EtherCATMasterState.TcDUT
TYPE ST_CX_EtherCATMasterState :
STRUCT
	arrADSAddr		: ARRAY[0..5] OF BYTE;
	nState			: UINT;
	nDevID			: UINT;
	nSlaveCount		: UINT;
	nDevState		: UINT;
END_STRUCT
END_TYPE

// ---- DUTs/METS/Device/CX Unit/EtherCAT/Terminal FBs/EBUS/ST_EBUS_AnalogueDataIn.TcDUT
TYPE ST_EBUS_AnalogueDataIn :
STRUCT
	nStatus		: WORD;
	nValue		: INT;
END_STRUCT
END_TYPE

// ---- DUTs/METS/Device/CX Unit/EtherCAT/Terminal FBs/EBUS/ST_EBUS_EtherCATState.TcDUT
TYPE ST_EBUS_EtherCATState :
STRUCT
	nState		: UINT;
	bWCState	: BOOL;
END_STRUCT
END_TYPE

// ---- DUTs/METS/Device/CX Unit/EtherCAT/Terminal FBs/KBUS/E_KBUS_RegisterAccessState.TcDUT
//{attribute 'qualified_only'}
//{attribute 'strict'}
TYPE E_KBUS_RegisterAccessState : (
	//E_KBUS_IDLE,
	//E_KBUS_REQUEST,
	//E_KBUS_RESPONSE,
	//E_KBUS_READREG,
	//E_KBUS_CHECKDATA,
	//E_KBUS_WRITEREG,
	//E_KBUS_RESETPROCESSDATA,
	//E_KBUS_PROCESSDATA,
	//E_KBUS_DONE
	E_KBUS_DUMMY
);
END_TYPE

// ---- DUTs/METS/Device/CX Unit/EtherCAT/Terminal FBs/KBUS/ST_KBUS_AnalogueDataIn.TcDUT
TYPE ST_KBUS_AnalogueDataIn :
STRUCT
	nState	: BYTE;
	nData	: INT;
END_STRUCT
END_TYPE

// ---- DUTs/METS/Device/CX Unit/EtherCAT/Terminal FBs/KBUS/ST_KBUS_AnalogueDataOut.TcDUT
TYPE ST_KBUS_AnalogueDataOut :
STRUCT
	nCtrl	: BYTE;
	nData	: INT;
END_STRUCT
END_TYPE

// ---- DUTs/METS/Device/CX Unit/EtherCAT/Terminal FBs/KBUS/ST_KBUS_KL1501DataIn.TcDUT
TYPE ST_KBUS_KL1501DataIn :
STRUCT
	nState	: BYTE;
	arrData	: ARRAY [0..1] OF UINT;
END_STRUCT
END_TYPE

// ---- DUTs/METS/Device/CX Unit/EtherCAT/Terminal FBs/KBUS/ST_KBUS_KL1501DataOut.TcDUT
TYPE ST_KBUS_KL1501DataOut :
STRUCT
	nCtrl	: BYTE;
	arrData	: ARRAY [0..1] OF UINT;
END_STRUCT
END_TYPE

// ---- DUTs/METS/Device/CX Unit/EtherCAT/Terminal FBs/KBUS/ST_KBUS_KL5001Config.TcDUT
TYPE ST_KBUS_KL5001Config :
STRUCT
	nTerminalType	: UINT;
	strFirmware		: STRING(2);
	nFeatureReg		: UINT;
	nDataRate		: UINT;		(* 1=MHz, 2=250kHz (default), 3=125kHz, 4=100kHz, 5=83kHz, 6=71kHz, 7=62.5kHz *)
	nDataBits		: UINT;		(* data bits (default=25) *)
END_STRUCT
END_TYPE

// ---- DUTs/METS/Device/CX Unit/EtherCAT/Terminal FBs/ST_EtherCATSlaveInfo.TcDUT
TYPE ST_EtherCATSlaveInfo :
STRUCT
	nAddr 			: UDINT;
	nlinkState		: UDINT;
	edeviceState	: ST_EcSlaveState;
	sType 			: STRING[16];
	sName 			: STRING[32];
END_STRUCT
END_TYPE

// ---- DUTs/METS/Device/CX Unit/EtherCAT/Terminal FBs/ST_EtherCATStatus.TcDUT
TYPE ST_EtherCATStatus :
STRUCT

	sEtherCATMasterAmsNetID	: T_AmsNetID;
	nSlavesCount				: UINT;
	arrSlaveInfo				: ARRAY[0..cMAX_ETHERCAT_SLAVES] OF ST_EtherCATSlaveInfo;
	nNodeWithError			: UINT;
	sNodeWithErrorName		: STRING(16);
END_STRUCT
END_TYPE

// ---- DUTs/METS/Device/CX Unit/Network/E_CX_NetworkInfoState.TcDUT
{attribute 'qualified_only'}
{attribute 'strict'}
TYPE E_CX_NetworkInfoState : (
	IDLE,
	GETDEVICETYPE,
	GETHOSTNAME,
	GETLOCALAMSNETID,
	GETADAPTERINFO,
	GETDNSINFO,
	GETSNTPSERVER,
	GETSNTPTIME,
	DONE
);
END_TYPE

// ---- DUTs/METS/Device/CX Unit/Network/E_CX_SetAMSNetIDState.TcDUT
{attribute 'qualified_only'}
{attribute 'strict'}
TYPE E_CX_SetAMSNetIDState : (
	//E_CX_SETAMSNETID_IDLE,
	//E_CX_SETAMSNETID_NEXTREGKEY,
	//E_CX_SETAMSNETID_READREGKEY,
	//E_CX_SETAMSNETID_WRITEREGKEY,
	//E_CX_SETAMSNETID_PAUSE,
	//E_CX_SETAMSNETID_REBOOT,
	//E_CX_SETAMSNETID_DONE
	DUMMY
);
END_TYPE

// ---- DUTs/METS/Device/CX Unit/Network/ST_CX_AdapterInfo.TcDUT
TYPE ST_CX_AdapterInfo :
STRUCT
	bDefault			: BOOL;
	strAdapterName		: STRING(75);
	bDHCPEnabled		: BOOL;
	strIPAddress		: T_IPv4Addr;
	strSubnetMask		: T_IPv4Addr;
	strDefaultGateway	: T_IPv4Addr;
END_STRUCT
END_TYPE

// ---- DUTs/METS/Device/CX Unit/Network/ST_CX_NetworkInfo.TcDUT
TYPE ST_CX_NetworkInfo :
STRUCT
	strDeviceName		: STRING(75);
	strAMSNetID			: STRING(23);
	strSNTPServer		: STRING(75);
	strSNTPRefreshTime	: STRING(31);
	arrAdapterInfo		: ARRAY[1..6] OF ST_CX_AdapterInfo;
END_STRUCT
END_TYPE

// ---- DUTs/METS/Device/CX Unit/NOVRAM/E_CX_NVDataCtrlState.TcDUT
{attribute 'qualified_only'}
{attribute 'strict'}
TYPE E_CX_NVDataCtrlState : (
	IDLE,
	PLATFORM,				(* initialisation *)
	DEVICEID,
	DEVICEINFO,
	READ,
	VALIDATE,
	COMPARE,				(* monitoring *)
	CHECKSUM,
	WRITE,
	EXPORT,
	IMPORT,
	OPENFILE,				(* export data *)
	ENCODEDATABLOCK,
	WRITEFILE,
	CLOSEFILE,
	READXMLDATA,		(* import data *)
	DECODEDATABLOCK,
	DONE := 20
);
END_TYPE

// ---- DUTs/METS/Device/CX Unit/NOVRAM/ST_CX_AMSAddress.TcDUT
TYPE ST_CX_AMSAddress :
STRUCT
	arrAMSNetID			: AMSNETID;
	nPortNo				: UINT;
END_STRUCT
END_TYPE

// ---- DUTs/METS/Device/CX Unit/NOVRAM/ST_CX_EL6080DataIn.TcDUT
TYPE ST_CX_EL6080DataIn :
STRUCT
	nStatus			: UINT;
	arrData			: ARRAY[0..1277] OF BYTE;
	bWcState		: BOOL;
	bInputToggle	: BOOL;
	nState			: UINT;
	sAMSAddress		: ST_CX_AMSAddress;
END_STRUCT
END_TYPE

// ---- DUTs/METS/Device/CX Unit/NOVRAM/ST_CX_EL6080DataOut.TcDUT
TYPE ST_CX_EL6080DataOut :
STRUCT
	nControl		: UINT;
	arrData			: ARRAY[0..1277] OF BYTE;
END_STRUCT
END_TYPE

// ---- DUTs/METS/Device/CX Unit/NOVRAM/ST_CX_NVDataBlock.TcDUT
TYPE ST_CX_NVDataBlock :
STRUCT
	DataOffs	: UDINT;
	Data		: STRING(2048);
END_STRUCT
END_TYPE

// ---- DUTs/METS/Device/CX Unit/System/E_CX_HWType.TcDUT
{attribute 'qualified_only'}
//{attribute 'strict'}
TYPE E_CX_HWType :
(
	//E_HW_UNKNOWN,
	CX1,
	CX2,
	CX5,
	CX8,
	CX9,
	CP,
	PC
);
END_TYPE

// ---- DUTs/METS/Device/Cylinders/E_CYLINDER_Position.TcDUT
{attribute 'qualified_only'}
{attribute 'strict'}
TYPE E_CYLINDER_Position :
(
	STOP		:= 0,
	EXTEND 		:= 1,
	RETRACT		:= 2
	//POSITION 	:=3
	
);
END_TYPE

// ---- DUTs/METS/Device/Cylinders/ST_CYLINDER_Control.TcDUT
TYPE ST_CYLINDER_Control :
STRUCT
	eCommand		: E_CYLINDER_Position;
END_STRUCT
END_TYPE

// ---- DUTs/METS/Device/Cylinders/ST_CYLINDER_IN.TcDUT
TYPE ST_CYLINDER_IN :
STRUCT
	bEnable				: BOOL;
	bRelExtend			: BOOL;
	bRelRetract			: BOOL;
END_STRUCT
END_TYPE

// ---- DUTs/METS/Device/Cylinders/ST_CYLINDER_OUT.TcDUT
TYPE ST_CYLINDER_OUT :
STRUCT
	bDeviceDisable					: BOOL;
	bMoveNotAllowed					: BOOL;

	bErrorPosition					: BOOL;
	bInPosition						: BOOL;
	bHomePosition					: BOOL;

	bCylinderInRetractedPosition	: BOOL;
	bCylinderInExtendedPosition		: BOOL;
	bCylinderIsRetracting			: BOOL;
	bCylinderIsExtending			: BOOL;

	stTagID							: ST_CYLINDER_TagID;

END_STRUCT
END_TYPE

// ---- DUTs/METS/Device/Cylinders/ST_CYLINDER_Status.TcDUT
 TYPE ST_CYLINDER_Status :
STRUCT

	I					: ST_CYLINDER_IN;
	Q					: ST_CYLINDER_OUT;

END_STRUCT
END_TYPE

// ---- DUTs/METS/Device/Cylinders/ST_CYLINDER_TagID.TcDUT
TYPE ST_CYLINDER_TagID :
STRUCT
	sDeviceTagID			: STRING(10);
	sRetractTagID			: STRING(10);
	sExtendTagID			: STRING(10);

END_STRUCT
END_TYPE

// ---- DUTs/METS/Device/DB/OLD/ST_DBResult.TcDUT
TYPE ST_DBResult :
STRUCT
	strCode : STRING(150);
	nExpiryStatus : DINT;
	(*nNumberOfchildren : INT;*)

(* nExpiryStatus:
0 - Expired
1 - Unknown - probaly due to reanimation. should still be successful
2 - Not Expired - OK*)
END_STRUCT
END_TYPE

// ---- DUTs/METS/Device/DB/OLD/ST_DB_CACCheckCtrl.TcDUT
TYPE ST_DB_CACCheckCtrl :
STRUCT
	bDB_ExecuteCacCheck			: BOOL;
	bDB_CACCheckComplete		: BOOL;
	bDB_CaseOk					: BOOL;
	bDB_Error						: BOOL;
	stCacToCheck					: ST_CAC_Data;
END_STRUCT
END_TYPE

// ---- DUTs/METS/Device/DB/OLD/ST_DB_Config.TcDUT
TYPE ST_DB_Config :
STRUCT

	bDBConfigured				: BOOL;
	sSQLName					: STRING;
	sDatabaseName				: STRING;
	stNetAddress				: ST_TCPIP_AddressPort;
	nLastDBID					: UDINT;

	bEnableOCVCheck							: BOOL;
	bEnableOACCheck							: BOOL;
	bEnableCACCheck							: BOOL;

END_STRUCT
END_TYPE

// ---- DUTs/METS/Device/DB/OLD/ST_DB_OACCheckCtrl.TcDUT
TYPE ST_DB_OACCheckCtrl :
STRUCT
	bDB_ExecuteOacCheck			: BOOL;
	bDB_OacCheckComplete			: BOOL;
	bOacValid						: BOOL;
	bDB_Error						: BOOL;
	stOacToCheck					: ST_OUTER_Status;
END_STRUCT
END_TYPE

// ---- DUTs/METS/Device/DB/OLD/ST_DB_OCVCheckCtrl.TcDUT
TYPE ST_DB_OCVCheckCtrl :
STRUCT
	bDB_ExecuteOcvCheck			: BOOL;
	bDB_OcvCheckComplete			: BOOL;
	bDB_AllCodesFound				: BOOL;
	bDB_Error						: BOOL;
	bDB_OCVValid					: BOOL;
	stOcvToCheck 					: ST_OUTER_Status;
END_STRUCT
END_TYPE

// ---- DUTs/METS/Device/DB/OLD/ST_DB_PcvCheckCtrl.TcDUT
TYPE ST_DB_PcvCheckCtrl :
STRUCT
	bDB_ExecutePcvCheck			: BOOL;
	bDB_PcvCheckComplete			: BOOL;
	bPackCodeFoundInDB			: BOOL;
	bPackExpired					: BOOL;
	sAssociatedCase 				: STRING(150);
	bDB_Error						: BOOL;
	stPackToCheck					: ST_PACK_Data;

END_STRUCT
END_TYPE

// ---- DUTs/METS/Device/DB/OLD/ST_DB_ReportDBCtrl.TcDUT
TYPE ST_DB_ReportDBCtrl :
STRUCT
	bExecuteCheck			: BOOL;
	bCheckComplete			: BOOL;
	sStoreProcedureName		: STRING := 'TC_DBReport';
	bDBError				: BOOL;
	nDBErrorID				: UDINT;
	sSqlState				: ST_DBSQLError;
	nRecords				: UDINT;
	stResultRecord			: ST_DB_ReportResult;

END_STRUCT
END_TYPE

// ---- DUTs/METS/Device/DB/OLD/ST_DB_ReportResult.TcDUT
TYPE ST_DB_ReportResult :
STRUCT
	nPackCodesTotal		: DINT;
	nPCV_NoDate 			: DINT;
	nPCV_NoOuterCode 	: DINT;
	nNoCACPack			: DINT;
	nOuterCodesTotal		: DINT;
	nOAC_NoDate 			: DINT;
	nNoOHMSuccesfull		: DINT;
	nNoCACOuter 			: DINT;
	nPackCodesArchive	 	: DINT;
	nOuterCodesArchive	: DINT;
END_STRUCT
END_TYPE

// ---- DUTs/METS/Device/DB/ST_DB_OACDataCtrl.TcDUT
TYPE ST_DB_OACDataCtrl :
STRUCT
	bCreateDataReq				: BOOL;	(* C *)
	bReadDataReq				: BOOL;	(* R *)
	bUpdateDataReq				: BOOL;	(* U *)
	bDeleteDataReq				: BOOL;	(* D *)

	sFileCodeName				: T_MaxString;
	
	bBlockRecord				: BOOL;
	bRestored					: BOOL;

	stOACStatusDB				: ST_OUTER_Status;

	bDone						: BOOL;
	bError						: BOOL;
	nErrorID					: UDINT;

END_STRUCT
END_TYPE

// ---- DUTs/METS/Device/DB/ST_DB_OCVDataCtrl.TcDUT
TYPE ST_DB_OCVDataCtrl :
STRUCT
	bCreateDataReq				: BOOL;	(* C *)
	bReadDataReq				: BOOL;	(* R *)
	bUpdateDataReq				: BOOL;	(* U *)
	bDeleteDataReq				: BOOL;	(* D *)

	sFileCodeName1				: T_MaxString;
	sFileCodeName2				: T_MaxString;
	
	bBlockRecord				: BOOL;
	bRestored					: BOOL;

	stOCVStatusDB				: ST_OUTER_Status;

	bDone						: BOOL;
	bError						: BOOL;
	nErrorID					: UDINT;

END_STRUCT
END_TYPE

// ---- DUTs/METS/Device/Drive/Analog/Config/ST_AnalogDrive.TcDUT
TYPE ST_AnalogDrive :
STRUCT
	nDriveSpeed					: INT:=60;
	tTimeOut						: TIME:=t#60s;
	(*bIsolatorExist					: BOOL;*)
	bBrakeExist					: BOOL:=TRUE;
	(*tBrakeDelayStart				: TIME:=t#100ms;*)
	tDriveDelayStart				: TIME:=t#500ms;
	(*tStoppingTime					: TIME:=t#10s;*)
END_STRUCT
END_TYPE

// ---- DUTs/METS/Device/Drive/Analog/ST_DriveCtrl.TcDUT
TYPE ST_DriveCtrl :
STRUCT
	bDriveRun:BOOL;
	nDriveAnalog:INT;
END_STRUCT
END_TYPE

// ---- DUTs/METS/Device/Drive/Analog/ST_PhtcCtrl.TcDUT
TYPE ST_PhtcCtrl :
STRUCT
	bStopInfeedConveyor:BOOL;
	bStopSeparator:BOOL;
END_STRUCT
END_TYPE

// ---- DUTs/METS/Device/Drive/MC2/Axis Control/ST_AXIS_Control.TcDUT
TYPE ST_AXIS_Control :
STRUCT
	eMotionType		: E_AXIS_MotionType;

	fDistance			: LREAL;	(*target relative position*)
	fPosition			: LREAL;	(*target absolute position*)
	fSetVelo			: LREAL;	(* target velocity *)
	bStopAtPos		: BOOL;	(* set TRUE to stop at specified pos, set FALSE to stop immediately *)
	fStopPos			: LREAL;	(* target modulo stop position *)

	bJogFwd			: BOOL;		(* set TRUE to jog forwards *)
	bJogRev			: BOOL;		(* set TRUE to jog reverse *)
	fJogVelo			: LREAL;	(* jog velocity (does not take effect if jog is in progress *)

END_STRUCT
END_TYPE

// ---- DUTs/METS/Device/Drive/MC2/Axis Control/ST_AXIS_IN.TcDUT
TYPE ST_AXIS_IN :
STRUCT
	bEnableAxis			: BOOL;
	bResetAxis		: BOOL;
	bHMIReleaseBreak	: BOOL;
	bEnableRevDir			: BOOL;		(* set TRUE to allow axis to run in reverse direction *)
	fOverride				: LREAL;	(* max axis output in % *)
	bFastStop			: BOOL;		(* set TRUE to override RUN signals and stop axis immediately *)
	bSafetyNotOK		: BOOL;
	nEtherCATState	: UINT;		(* EtherCAT operating state *)

END_STRUCT
END_TYPE

// ---- DUTs/METS/Device/Drive/MC2/Axis Control/ST_AXIS_OUT.TcDUT
TYPE ST_AXIS_OUT :
STRUCT

	bInitOK				: BOOL;		(* TRUE = parameter set read at least once *)
	bEnabled			: BOOL;		(* TRUE = axis is enabled *)
	bActive				: BOOL;		(* TRUE = axis is moving *)
	bHomeActive			: BOOL;
	bVeloActive			: BOOL;
	bAbsActive			: BOOL;
	bRelActive			: BOOL;
	bJogActive			: BOOL;		(* TRUE = axis is moving in JOG mode *)
	bRunningFwd			: BOOL;		(* TRUE = axis is running forwards *)
	bRunningRev			: BOOL;		(* TRUE = axis is running backwards *)
	bCalibrated			: BOOL;		(*TRUE = axis has benn calibrated*)
	(*bHomed				: BOOL;*)		(* TRUE = axis has been homed *)
	bAxisError			: BOOL;		(* TRUE = axis is in error state *)
	nAxisErrorID		: UDINT;	(* NC axis error code *)
	fActPos				: LREAL;	(* axis absolute position *)
	fModuloPos			: LREAL;	(* axis modulo position *)
	fActVelo			: LREAL;	(* axis act ual velocity *)
	bDriveError			: BOOL;		(* TRUE = drive is in error state *)
	nStatusDWord		: DWORD;	(* drive status code *)
	fAmplifierTemp		: LREAL;	(* Amplifier temperature (degrees) *)
	fDCLinkVolts		: LREAL;	(* DC link voltage (volts) *)

END_STRUCT
END_TYPE

// ---- DUTs/METS/Device/Drive/MC2/Axis Control/ST_AXIS_Status.TcDUT
 TYPE ST_AXIS_Status :
STRUCT

	I					: ST_AXIS_IN;
	Q					: ST_AXIS_OUT;

END_STRUCT
END_TYPE

// ---- DUTs/METS/Device/Drive/MC2/Config/ST_AXIS_Config.TcDUT
TYPE ST_AXIS_Config :
STRUCT

	sDeviceName				: STRING(30) := 'Axis';
	bCalibrationSensorExist	: BOOL;
	nTorqueLimitation			: UINT	:=	32767;
	stRamps					: ST_AxisCtrlRamps;

END_STRUCT
END_TYPE

// ---- DUTs/METS/Device/Drive/MC2/EtherCAT/AX5000 FBs/ST_AX5000_TouchProbe.TcDUT
TYPE ST_AX5000_TouchProbe :
STRUCT
	nStatusWord		: UINT;
	nHardCounts		: DINT;
	nPosEdge		: DINT;
	nNegEdge		: DINT;
END_STRUCT
END_TYPE

// ---- DUTs/METS/Device/Drive/MC2/EtherCAT/Encoder FBs/ST_DeviceAddress.TcDUT
TYPE ST_DeviceAddress :
STRUCT
	arrNetID		: ARRAY[0..5] OF BYTE;
	nPortNo			: UINT;
END_STRUCT
END_TYPE

// ---- DUTs/METS/Device/Drive/MC2/NC Axis/E_AXIS_CtrlState.TcDUT
{attribute 'qualified_only'}
{attribute 'strict'}
TYPE E_AXIS_CtrlState : (
	IDLE,
	JOG,
	MOVEVELO1,
	MOVEVELO2,
	MOVERELATIVE,
	MOVEABSOLUTE,
	//E_AXIS_HOMINGPOS,
	STOPPOS,
	HALT,
	FASTSTOP
);
END_TYPE

// ---- DUTs/METS/Device/Drive/MC2/NC Axis/E_TORQUE_Scaling.TcDUT
//{attribute 'qualified_only'}
//{attribute 'strict'}
TYPE E_TORQUE_Scaling : (
	//E_TORQUE_IDLE,
	//E_TORQUE_GETPORTNO,
	//E_TORQUE_RATEDCURRENT,
	//E_TORQUE_MAXCURRENT,
	//E_TORQUE_MONITOR,
	//E_TORQUE_ERROR,
	E_TORQUE_DUMMY
);
END_TYPE

// ---- DUTs/METS/Device/Drive/MC2/NC Axis/ST_AxisCtrlRamps.TcDUT
TYPE ST_AxisCtrlRamps :
STRUCT
	fFastStopDecel	: LREAL;
	fFastStopJerk	: LREAL;
	fNormalAccel	: LREAL;
	fNormalDecel	: LREAL;
	fNormalJerk		: LREAL;
	fJogAccel		: LREAL;
	fJogDecel		: LREAL;
	fJogJerk		: LREAL;
END_STRUCT
END_TYPE

// ---- DUTs/METS/Device/Drive/MC2/NC Axis/ST_DriveStatus.TcDUT
TYPE ST_DriveStatus :
STRUCT
	nActLength	: UINT;
	nMaxLength	: UINT;
	strStatus	: STRING;
END_STRUCT
END_TYPE

// ---- DUTs/METS/Device/Drive/MC2/NC Axis/ST_LatchPosBuffer.TcDUT
TYPE ST_LatchPosBuffer :
STRUCT
	nIndex			: BYTE;		(* index of arrLatchedPos where last value was added *)
	bBufferHasData	: BOOL;		(* indicates buffer has 1 or more values in arrLatchedPos *)
	bPosAdded		: BOOL;		(* set TRUE for 1 cycle when new value has been added to arrLatchedPos *)
	bPosDeleted		: BOOL;		(* set TRUE for 1 cycle when new value has been deleted from arrLatchedPos *)
	fLastTargetPos	: LREAL;	(* last position removed from arrLatchedPos *)
	fLastFeedLength	: LREAL;	(* distance moved to reach fLastTargetPos *)
	fNextFeedLength	: LREAL;	(* distance to move from fLastTargetPos to arrLatchedPos[1] *)
	arrLatchedPos	: ARRAY[1..25] OF LREAL;	(* array of latched position values *)
END_STRUCT
END_TYPE

// ---- DUTs/METS/Device/Drive/MC2/NC Axis/ST_NC_EncDataIn.TcDUT
TYPE ST_NC_EncDataIn :
STRUCT
	nInData1	: ARRAY[0..1] OF UINT;
	nInData2	: ARRAY[0..1] OF UINT;
	nStatus1	: BYTE;
	nStatus2	: BYTE;
	nStatus3	: BYTE;
	nStatus4	: BYTE;
END_STRUCT
END_TYPE

// ---- DUTs/METS/Device/Drive/MC2/NC Axis/ST_NC_EncDataOut.TcDUT
TYPE ST_NC_EncDataOut :
STRUCT
	nOutData1	: ARRAY[0..1] OF UINT;
	nOutData2	: ARRAY[0..1] OF UINT;
	nCtrl1		: BYTE;
	nCtrl2		: BYTE;
	nCtrl3		: BYTE;
	nCtrl4		: BYTE;
END_STRUCT
END_TYPE

// ---- DUTs/METS/Device/Drive/MC2/TempAxis/ST_AxisHomeStruct.TcDUT
TYPE ST_AxisHomeStruct :
STRUCT

	n_State								: 	DINT;			(* Current Sequence State *)
	n_StateBuffer							: 	DINT;			(* Next Sequence State *)
	b_FunctionRequest						: 	BOOL;		(* Sequence Function Request from Home *)
	b_FunctionInProgress					: 	BOOL;		(* Sequence Function In Progress Handshaking *)
	b_FunctionComplete					: 	BOOL;		(* Sequence Function Complete Handshaking *)
	b_FunctionAbort						: 	BOOL;		(* Sequence Function Abort *)
	b_FunctionHomed						: 	BOOL;		(* Sequence Function Homed *)
	b_CycleStopped						: 	BOOL;		(* Sequence Function Cycle Stopped *)
	n_Handshaking							: 	DINT;		(* Generic Handshaking Tag *)
	b_AxisHome							:	BOOL;
	b_AxisStop							:	BOOL;
	b_MoveToEndStop						:	BOOL;
	b_AxisEnable							:	BOOL;
	b_AxisReset							:	BOOL;

END_STRUCT
END_TYPE

// ---- DUTs/METS/Device/Drive/MC2/TempAxis/ST_AxisMotionStruct.TcDUT
TYPE ST_AxisMotionStruct :
STRUCT

	n_State 								: 	DINT;		(* Current Sequence State *)
	n_StateBuffer							: 	DINT;		(* Next Sequence State *)
	b_FunctionRequest						: 	BOOL;		(* Sequence Function Request from Home *)
	b_FunctionInProgress					: 	BOOL;		(* Sequence Function In Progress Handshaking *)
	b_FunctionComplete					: 	BOOL;		(* Sequence Function Complete Handshaking *)
	b_FunctionAbort						: 	BOOL;		(* Sequence Function Abort *)
	b_FunctionHomed						: 	BOOL;		(* Sequence Function Homed *)
	b_CycleStopped						: 	BOOL;		(* Sequence Function Cycle Stopped *)
	n_Handshaking							: 	DINT;		(* Generic Handshaking Tag *)
	b_AxisMoveVelocity						:	BOOL;
	b_AxisMoveRelative						: 	BOOL;
	b_AxisMoveModulo				  		: 	BOOL;
	b_MoveToP0							:	BOOL;
	b_MoveToP02							:	BOOL;
	b_MoveP0_P1							:	BOOL;
	b_MoveP1_P0							:	BOOL;
	b_MoveP1_P2							:	BOOL;
	b_MoveP2_P3							:	BOOL;
	b_MoveP2_P0							:	BOOL;
	b_MoveP3_P0							:	BOOL;
	b_MoveP3_P4							:	BOOL;
	b_Move_IDPos							:	BOOL;
	b_AxisEnable							:	BOOL;
	b_AxisReset							:	BOOL;
	b_AtP1								:	BOOL;
	b_AtP2								:	BOOL;
	b_AtP3								:	BOOL;
	b_AtP4								:	BOOL;
	b_AtP1TimerComplete					:	BOOL;
	b_AtVelocity1							:	BOOL;
	b_ExtendEject							:	BOOL;
	b_HomeRequired						:	BOOL;
	b_OKToIndex							:	BOOL;
	b_Referenced							:	BOOL;
	b_AxisHome							:	BOOL;
	b_AxisStop							:	BOOL;
	b_MoveToEndStop						:	BOOL;
	b_MandrelID_OK						:	BOOL;
	b_IDRequest							:	BOOL;
	b_IDInProgress							:	BOOL;
	b_IDComplete							:	BOOL;

END_STRUCT
END_TYPE

// ---- DUTs/METS/Device/Drive/Profinet/Config/ST_ProfinetDrive.TcDUT
TYPE ST_ProfinetDrive :
STRUCT
	bEnable									: BOOL;
	sDeviceName								: STRING(30) := 'Drive';
	cuiProfinetPortofDrive						: UINT:=4125;
	etDriveReference                      			: INT := 1;
	cusiDriveID								: USINT:=1;
	(*ctTimeOut								: TIME:=T#5S;*)
	bBrakeExist								: BOOL:=TRUE;

	tRumpUpTime								: TIME := t#250ms;
	nDriverSpeedHz 							: UINT :=50;
	tDriveDelayStart							: TIME :=t#100ms;
	tDriverOffDelay							: TIME :=t#3s;

	fSpeedScalefactor							: REAL := 140;
	fTorqueScaleFactor						: REAL := 120.48;
	nTorqueLimit								: REAL := 1;

	fReferenceSpeedFrequencyP2000			: REAL := 3000;
	fReferenceCurrentP2002					: REAL := 5;
	fReferenceTorqueP2003					: REAL := 5;

END_STRUCT
END_TYPE

// ---- DUTs/METS/Device/Drive/Profinet/Config/ST_ProfinetMasterConfig.TcDUT
TYPE ST_ProfinetMasterConfig :
(* EL6631 *)
STRUCT
	strTAMSNETID_ProfinetMasterEthercatAmsNetId			: T_AmsNetId:=''; (* string(23) *)
	strIPAddress										: STRING(15) := ''; (* currently display only not linked *)

END_STRUCT
END_TYPE

// ---- DUTs/METS/Device/Drive/Profinet/E_DRIVE_Name.TcDUT
{attribute 'qualified_only'}
{attribute 'strict'}
TYPE E_DRIVE_Name :
(
	OUTER_SEPAR			:=1,	(*PAOL*)
	INFEED_CONV			:=2,	(*CML*)
	ROTARY_TRNSFR		:=3,	(*CML*)
	LOWR_BELTS			:=4,	(*CML*)
	REJECT_CONV			:=5,	(*CML*)
	TRANSF_CONV			:=6,	(*SFLX*)
	ADDIT_CONV			:=7,	(*MM*)
	OUTFD_CONV			:=8		(*SFLX*)

);
END_TYPE

// ---- DUTs/METS/Device/Drive/Profinet/Parameters/ST_DataPntAdr.TcDUT
TYPE ST_DataPntAdr :
STRUCT
	pAddress		:UDINT;
	udiSize		:UDINT;
END_STRUCT
END_TYPE

// ---- DUTs/METS/Device/Drive/Profinet/Parameters/ST_KeyPadDisplay.TcDUT
TYPE ST_KeyPadDisplay :
STRUCT
	sTopLine                         :STRING[12];
    	sTopLineUnit                  :STRING[5];
   	rBottomLine                     :REAL;
    	sBottomLineUnit            :STRING[5];
END_STRUCT
END_TYPE

// ---- DUTs/METS/Device/Drive/Profinet/Parameters/ST_Parameter.TcDUT
TYPE ST_Parameter :
STRUCT
	   uiParameter     	:UINT;
	   uiSubIndex      	:UINT;
	   stValue         		:ST_Value;
	   sString         		:STRING[30];
	   eFormat     		:E_PD_Datatype;
	   (*IEC 61158-5: Fieldbus data types specify the machine independent syntax FOR application data 
		conveyed BY FAL services. A certain set OF common data types is standardized FOR PROFIBUS DP AND 
		has an assigned data TYPE numeric identifier. Following some frequently occurring data types AND IDs:
		1    Boolean                6    Unsigned16
		2    Integer8               7    Unsigned32
		3    Integer16              8    Floating point
		4    Integer32              9    Visible STRING
		5    Unsigned8              10   Octet STRING
                *)
END_STRUCT
END_TYPE

// ---- DUTs/METS/Device/Drive/Profinet/Parameters/ST_ParameterControl.TcDUT
TYPE ST_ParameterControl :
STRUCT
	etDriveReference                      	:INT;
           xHMIDriveDownButton                   :BOOL;
           xHMIDriveUpButton                     	:BOOL;
           xRefreshButton                       		:BOOL;
           xWriteParametersButton             	:BOOL;
           stHMIStandardReadParameters           	:ST_Parameters;
           stHMIStandardReadWriteParameters      	:ST_Parameters;
           stHMIFastReadParameterList           		:ST_Parameters;
           iHMIReadSequence                      			:INT;
           stKeyPadDisplay                      			:ST_KeyPadDisplay;
           udiAdvancedParameter                  		:UDINT;(*Advanced Parameter*)
           udiAdvancedSubIndex                   		:UDINT;(*Advanced Sub Index Parameter*)
	  etDataType							:INT;
           etDrivesAvailable                     			:INT;
           etServosAvailable                      			:INT;
           xLoading                               				:BOOL;
END_STRUCT
END_TYPE

// ---- DUTs/METS/Device/Drive/Profinet/Parameters/ST_Parameters.TcDUT
TYPE ST_Parameters :
STRUCT
	astParameterList                :ARRAY[1..cPARAMETER_STORAGE_SIZE]OF ST_Parameter;
END_STRUCT
END_TYPE

// ---- DUTs/METS/Device/Drive/Profinet/Parameters/ST_Value.TcDUT
TYPE ST_Value :
STRUCT
	xValueType1             	:BOOL;
	siValueType2            	:SINT;
	iValueType3             	:INT;
	diValueType4            	:DINT;
	usiValueType5           	:USINT;
	uiValueType6            	:UINT;
	udiValueType7           	:UDINT;
	rValueType8                 	:REAL;
	sValueType9                 	:STRING;
END_STRUCT
END_TYPE

// ---- DUTs/METS/Device/Drive/Profinet/ST_PNetMasterStatus.TcDUT
TYPE ST_PNetMasterStatus :
(* EL6631 *)
STRUCT
	nPNetIoError		: UINT;
	nPNetIoDiag		: UINT;
END_STRUCT
END_TYPE

// ---- DUTs/METS/Device/Drive/Profinet/_G120/Drives/E_DRIVE_DataType.TcDUT
//{attribute 'qualified_only'}
//{attribute 'strict'}
TYPE E_DRIVE_DataType :
(*
Version history:
Date		|	Version/Author 		|	Remark
----------------------------------------------------------------------------------------------------
09.02.18	|	2.000.016	PSA		|	Original Version.
									|	Siemens G120 drive data type enumerations
*)
(
	//eNull, 
	//eBool, 
	//eInt, 
	//eDInt, 
	//eFloat
	eDUMMY
);
END_TYPE

// ---- DUTs/METS/Device/Drive/Profinet/_G120/Drives/ST_DRIVE_INPUT.TcDUT
TYPE ST_DRIVE_INPUT :
	(*
Version history:
Date		|	Version/Author 		|	Remark
----------------------------------------------------------------------------------------------------
09.02.18	|	2.000.016	PSA		|	Original Version.
									|	Siemens G120 drive IO input structure
*)
STRUCT
	uiDriveInput					: ARRAY[1..10] OF UINT;
END_STRUCT
END_TYPE

// ---- DUTs/METS/Device/Drive/Profinet/_G120/Drives/ST_DRIVE_OUTPUT.TcDUT
TYPE ST_DRIVE_OUTPUT :
(*
Version history:
Date		|	Version/Author 		|	Remark
----------------------------------------------------------------------------------------------------
09.02.18	|	2.000.016	PSA		|	Original Version.
									|	Siemens G120 drive IO output structure
*)
STRUCT
	uiDriveOutput						: ARRAY[1..10] OF UINT;
END_STRUCT
END_TYPE

// ---- DUTs/METS/Device/Drive/Profinet/_G120/Drives/ST_DRIVE_STATUS.TcDUT
TYPE ST_DRIVE_STATUS :
(*
Version history:
Date		|	Version/Author 		|	Remark
----------------------------------------------------------------------------------------------------
09.02.18	|	2.000.016	PSA		|	Original Version.
									|	Siemens G120 drive status infomaration structure
*)
STRUCT
	xReadyForSwitchingOn	: BOOL;
	xReady					: BOOL;
	xOperationEnable		: BOOL;
	xPowerOnInhibit			: BOOL;
	xFault					: BOOL;
	xAlarm					: BOOL;
	xTorqueLimitReached		: BOOL;
	xSpeedExceeded			: BOOL;
	xHoldingBrake			: BOOL;
	xMotorOverTemp			: BOOL;
	xMotorRotatingClockwise	: BOOL;
	xMotorRotatingCClockwise: BOOL;
	xControlRequested		: BOOL;
	xSetSpeedPointReached	: BOOL;

	rActualSpeed			: REAL;
	rCurrent				: REAL;
	rTorque					: REAL;
	iWarningCode			: UINT;
	iFaultCode				: UINT;
END_STRUCT
END_TYPE

// ---- DUTs/METS/Device/Drive/Profinet/_G120/Drives/ST_G120_ExtendedIn.TcDUT
TYPE ST_G120_ExtendedIn :
(*
Version history:
Date		|	Version/Author 		|	Remark
----------------------------------------------------------------------------------------------------
09.02.18	|	2.000.016	PSA		|	Original Version.
									|	Siemens G120 drive extended input structure
*)
STRUCT
	rSpeedScalefactor				: REAL := 140;
	rTorqueScaleFactor				: REAL := 120.48;
	uiTorqueLimit					: UINT;
	rReferenceSpeedFrequencyP2000	: REAL := 3000;
	rReferenceCurrentP2002			: REAL := 5;
	rReferenceTorqueP2003			: REAL := 5;
	tRumpUpTime						: TIME := t#1s;
	uiParameter						: UINT;
	uiIndex							: UINT;
	eParameterType					: E_DRIVE_DataType;
	xValue							: BOOL;
	iValue							: INT;
	diValue							: DINT;
	rValue							: REAL;
END_STRUCT
END_TYPE

// ---- DUTs/METS/Device/Drive/Profinet/_G120/Drives/ST_G120_ExtendedOut.TcDUT
TYPE ST_G120_ExtendedOut :
(*
Version history:
Date		|	Version/Author 		|	Remark
----------------------------------------------------------------------------------------------------
09.02.18	|	2.000.016	PSA		|	Original Version.
									|	Siemens G120 drive extended output structure
*)
STRUCT
	xTorqueLimitReached				: BOOL;
	xSpeedExceeded					: BOOL;
	xHoldingBrake					: BOOL;
	xMotorOverTemp					: BOOL;
	xMotorRotatingClockwise			: BOOL;
	xMotorRotatingCClockwise		: BOOL;
	xControlRequested				: BOOL;
	xSetSpeedPointReached			: BOOL;

	xValue							: BOOL;
	iValue							: INT;
	diValue							: DINT;
	rValue							: REAL;
	xReadWriteError					: BOOL;
	uiFaultCode						: UINT;
END_STRUCT
END_TYPE

// ---- DUTs/METS/Device/Drive/Profinet/_G120/Drives/ST_G120_IN.TcDUT
TYPE ST_G120_IN :
(*
Version history:
Date		|	Version/Author 		|	Remark
----------------------------------------------------------------------------------------------------
09.02.18	|	2.000.016	PSA		|	Original Version.
									|	Siemens G120 drive control input structure
*)
STRUCT
	xEnable							: BOOL;
	xDriveEnable					: BOOL;
	xClearFault						: BOOL;
	xInvertDirection				: BOOL;
	uiSpeed							: UINT;
	stExt							: ST_G120_ExtendedIn;
END_STRUCT
END_TYPE

// ---- DUTs/METS/Device/Drive/Profinet/_G120/Drives/ST_G120_Status.TcDUT
TYPE ST_G120_Status :
(*
Version history:
Date		|	Version/Author 		|	Remark
----------------------------------------------------------------------------------------------------
09.02.18	|	2.000.016	PSA		|	Original Version.
									|	Siemens G120 drive structure
*)
STRUCT
	I								: ST_G120_IN;
	Q								: ST_G120_OUT;
END_STRUCT
END_TYPE

// ---- DUTs/METS/Device/Drive/Profinet/_G120/ST_G120_Control.TcDUT
TYPE ST_G120_Control :
STRUCT
	bSafetyOk			: BOOL;
	bRun				: BOOL;
	bClearFault			: BOOL;
	nSpeedHz 			: UINT;
	bInvertDirection		: BOOL;
END_STRUCT
END_TYPE

// ---- DUTs/METS/Device/Encoders/CAMS/ST_AFS60_Cam.TcDUT
TYPE ST_AFS60_Cam :
STRUCT
	bEnable				: BOOL;
	nLowerLimit1		: UDINT;
	nLowerLimit2		: UDINT;
	nUpperLimit1		: UDINT;
	nUpperLimit2		: UDINT;
END_STRUCT
END_TYPE

// ---- DUTs/METS/Device/Encoders/CAMS/ST_AFS60_CamHMi.TcDUT
TYPE ST_AFS60_CamHMi :
STRUCT
	bEnable				: BOOL;
	fLowerLimit1		: LREAL; (* channel 1 *)
	fLowerLimit2		: LREAL; (* channel 2 *)
	fUpperLimit1		: LREAL;
	fUpperLimit2		: LREAL;
	fRange				: LREAL := 360.0;
	sDesciption			: STRING := 'Cam';
END_STRUCT
END_TYPE

// ---- DUTs/METS/Device/Encoders/CAMS/ST_AFS60_Config.TcDUT
TYPE ST_AFS60_Config :
STRUCT
		nCamScallingFactor				: LREAL := 0.001373291015625; (* cound per degree  *)
		stCamsHMi						: ARRAY[1..8] OF ST_AFS60_CamHMi; (* 8 in encoder *)
		nEncoderSlaveAddress			: UINT := 1025; (* ethercat slave address. Ethercat tab -> Ethercat Addr *)
		nEncoderPresetZero				: UDINT;
		strCAMDeviceName				: STRING := 'Device 1 (EtherCAT)';
		strCAMBoxName				: STRING := 'CAM1 (SICK AFS60A ST, 18-Bit)';
END_STRUCT
END_TYPE

// ---- DUTs/METS/Device/Encoders/CAMS/ST_AFS60_Status.TcDUT
TYPE ST_AFS60_Status :
STRUCT
	fActualValue					: LREAL;
	fTemp							: LREAL;
	nMsecUpTime					: UDINT;
	bCam1							: BOOL;
	bCam2							: BOOL;
	bCam3							: BOOL;
	bCam4							: BOOL;
	bCam5							: BOOL;
	bCam6							: BOOL;
	bCam7							: BOOL;
	bCam8							: BOOL;
END_STRUCT
END_TYPE

// ---- DUTs/METS/Device/Encoders/ST_ENCODER_IN.TcDUT
 TYPE ST_ENCODER_IN :
STRUCT
	bEnable				: BOOL;
END_STRUCT
END_TYPE

// ---- DUTs/METS/Device/Encoders/ST_ENCODER_OUT.TcDUT
TYPE ST_ENCODER_OUT :
STRUCT
	bDeviceDisable			: BOOL;

	nRevolutions			: UDINT := 0;
	nPulses				: UDINT;
	fPositionInMM			: LREAL;

	bError					: BOOL;
	sError					: STRING;

	nWarningStatus		: UINT;
	nAlarmStatus			: UINT;

END_STRUCT
END_TYPE

// ---- DUTs/METS/Device/Encoders/ST_ENCODER_Status.TcDUT
  TYPE ST_ENCODER_Status :
STRUCT

	I					: ST_ENCODER_IN;
	Q					: ST_ENCODER_OUT;

END_STRUCT
END_TYPE

// ---- DUTs/METS/Device/IO2 Controls/E_IO2_InputSource.TcDUT
{attribute 'qualified_only'}
{attribute 'strict'}
TYPE E_IO2_InputSource :
(
	SENSOR	:= 1,
	MACHINE := 2
);
END_TYPE

// ---- DUTs/METS/Device/IO2 Controls/E_IO2_Type.TcDUT
{attribute 'qualified_only'}
{attribute 'strict'}
TYPE E_IO2_Type :
(
	BLOCKED	:= 0,
	NO := 1,
	NC := 2
);
END_TYPE

// ---- DUTs/METS/Device/IO2 Controls/Input Ctrl/ST_IO2_DoubleInputCtrl.TcDUT
TYPE ST_IO2_DoubleInputCtrl :
STRUCT
	eInputSource			: E_IO2_InputSource;
	sInputName			: STRING(40);

	eTypeInput1			: E_IO2_Type;
	tTimeOnFilter1			: TIME;
	tTimeOffFilter1			: TIME;

	eTypeInput2			: E_IO2_Type;
	tTimeOnFilter2			: TIME;
	tTimeOffFilter2			: TIME;
END_STRUCT
END_TYPE

// ---- DUTs/METS/Device/IO2 Controls/Input Ctrl/ST_IO2_DoubleInputLockedCtrl.TcDUT
TYPE ST_IO2_DoubleInputLockedCtrl :
STRUCT
	eInputSource			: E_IO2_InputSource;
	sInputName		: STRING(40);

	eTypeInput1			: E_IO2_Type;
	tTimeOnFilter1			: TIME;
	tTimeOffFilter1			: TIME;
	tTimeLatch1			: TIME;

	eTypeInput2			: E_IO2_Type;
	tTimeOnFilter2			: TIME;
	tTimeOffFilter2			: TIME;
	tTimeLatch2			: TIME;
END_STRUCT
END_TYPE

// ---- DUTs/METS/Device/IO2 Controls/Input Ctrl/ST_IO2_SingleInputCtrl.TcDUT
TYPE ST_IO2_SingleInputCtrl :
STRUCT
	eTypeInput 		: E_IO2_Type;
	tTimeOnFilter		: TIME;
	tTimeOffFilter 		: TIME;
	sInputName		: STRING(40);
END_STRUCT
END_TYPE

// ---- DUTs/METS/Device/IO2 Controls/Input Ctrl/ST_IO2_SingleInputLockedCtrl.TcDUT
TYPE ST_IO2_SingleInputLockedCtrl :
STRUCT
	eTypeInput 		: E_IO2_Type;
	tTimeOnFilter		: TIME;
	tTimeOffFilter 		: TIME;
	tTimeLatch			: TIME;
	sInputName		: STRING(40);
END_STRUCT
END_TYPE

// ---- DUTs/METS/Device/IO2 Controls/Outpout Ctrl/ST_IO2_OutputCtrl.TcDUT
TYPE ST_IO2_OutputCtrl :
STRUCT
	eTypeOutput		: E_IO2_Type;
	tOutputDelayed	: TIME;
	tOutputLocked		: TIME;
	sOutputName		: STRING(40);
END_STRUCT
END_TYPE

// ---- DUTs/METS/Device/IO2 Controls/ST_IO2_Diagnostic.TcDUT
TYPE ST_IO2_Diagnostic :
STRUCT
	bState		: BOOL;
	sVarName		: STRING;

END_STRUCT
END_TYPE

// ---- DUTs/METS/Device/IO2 Controls/ST_IO2_InputPLC.TcDUT
TYPE ST_IO2_InputPLC :
STRUCT
	bRawInput			: BOOL;
	bRawRTrigger			: BOOL;
	bRawFTrigger			: BOOL;
	bStateInput			: BOOL;
	bStateRTrigger			: BOOL;
	bStateFTrigger			: BOOL;
END_STRUCT
END_TYPE

// ---- DUTs/METS/Device/IO2 Controls/ST_IO2_OutputPLC.TcDUT
TYPE ST_IO2_OutputPLC :
STRUCT
	bOutputEnable				: BOOL;

	bStateOutput				: BOOL;
	bDelayedOutput			: BOOL;
	bLockedOutput			: BOOL;
	bDelayedLockedOtput		: BOOL;
END_STRUCT
END_TYPE

// ---- DUTs/METS/Device/Printers/E_PRINTER_State.TcDUT
{attribute 'qualified_only'}
{attribute 'strict'}
TYPE E_PRINTER_State :
(
	IDLE,
	//E_PRINTER_CONNECT,
	//E_PRINTER_COMMAND,
	SEND,
	RECEIVE,
	//E_PRINTER_LOADDATA,
	//E_PRINTER_FILESIZE,
	DISCONNECT,
	DONE
);
END_TYPE

// ---- DUTs/METS/Device/Printers/ST_PRINTER_Config.TcDUT
TYPE ST_PRINTER_Config :
STRUCT

	bEnable				: BOOL;
	sDeviceName			: STRING(30) := 'Printer';
	sPrinterID				: STRING;							(*Printer ID, used to request the correct codes from the database*)

	stIPAdressPort			:  ST_TCPIP_AddressPort;
	tTimeout				: TIME;			(* TCP command timeout delay *)

END_STRUCT
END_TYPE

// ---- DUTs/METS/Device/Printers/ST_PRINTER_IN.TcDUT
TYPE ST_PRINTER_IN :
STRUCT

	bSystemReset			: BOOL;			(* set TRUE to send SystemReset command to printer *)
	bSendCommand		: BOOL;			(* set TRUE to send command to printer *)
	sCommand				: T_LongSTRING;	(* command to be sent to the printer *)

END_STRUCT
END_TYPE

// ---- DUTs/METS/Device/Printers/ST_PRINTER_OUT.TcDUT
TYPE ST_PRINTER_OUT :
STRUCT

	bPrinterReady		: BOOL;			(* TRUE = printer comms OK *)
	bSystemResetOK		: BOOL;			(* TRUE = system reset command sent to printer *)
	nStatusCode			: INT;			(* printer status code *)
	sResponse			: STRING(255);	(* command response string *)
	sCurrentCode					: STRING(255);
	(*aLast10CodesPrinted				: ARRAY[1..10] OF STRING(255);*)
	eSocketState		: E_SocketConnectionState;	(* TCP socket connection state *)

END_STRUCT
END_TYPE

// ---- DUTs/METS/Device/Printers/ST_PRINTER_Status.TcDUT
(*
Version history:
Date		|	Version/Author 		|	Remark
----------------------------------------------------------------------------------------------------
14.09.16	|	1.000.001	PSA		|	Original Version.
									|	Printer data structure
*)
TYPE ST_PRINTER_Status :
STRUCT

(* read only *)
	bPrinterReady					: BOOL;
	bActivePrinter					: BOOL;
	bPrinterInService				: BOOL;		(*printer Avalable*)
	bDataReady					: BOOL;
	bHomePosition				: BOOL;
	bLabelPrinted					: BOOL;
	bReadyToApply				: BOOL;
	bApplyDone					: BOOL;
	bSummaryWarning				: BOOL;
	bPrinterError					: BOOL;

	bSelectPrinter					: BOOL;
	bPrinterSelected				: BOOL;

	I					: ST_PRINTER_IN;
	Q					: ST_PRINTER_OUT;

	aLast10CodesPrinted	: ARRAY[1..10] OF T_OUTER_Barcode;


	(*nPrinterStatusCode			: INT;
	nPrinterState					: BYTE;
	eLabelStatus					: E_WOLKE_LABEL_STATUS;
	ePrintLabelStatus				: E_WOLKE_PRINT_LABEL_STATUS;
	ePLabelStatus					: E_WOLKE_PLABEL_STATUS;
	strInkLevel						: STRING;
	sManualCtrlPrinter				: ST_PRINTER_ManualCtrl;
	sCurrentCode					: STRING(255);
	aLastPrintedCodes				: ARRAY[1..10] OF STRING(255);
	eSocketState					: E_SocketConnectionState;*)

END_STRUCT
END_TYPE

// ---- DUTs/METS/Device/Scanner/E_SCANNER_CodeType.TcDUT
{attribute 'qualified_only'}
//{attribute 'strict'}
TYPE E_SCANNER_CodeType :
(
	NONE 		:= 0,
	OCR			:= 7,
	DATAMARTIX	:= 10,
	QR			:= 11,
	DOTCODE		:= 14,
	CODE128		:= 20,
	ITF14		:= 24,
	EAN13		:= 27,
	EAN8		:= 28,
	UNKNOWN		:= 99
);
END_TYPE

// ---- DUTs/METS/Device/Scanner/E_SCANNER_DeviceType.TcDUT
{attribute 'qualified_only'}
//{attribute 'strict'}
TYPE E_SCANNER_DeviceType :    (*tAcquisitionTime - to be secured*)
(
	NONE,
	MV420_F,			//F -> Full resolution
	MV420_H,			//H -> Half resolution
	MV440SR_F,
	MV440SR_H,
	MV440HR_F,
	MV440HR_H,
	MV440UR_F,
	MV440UR_H,
	MV540S_F,
	MV540S_H,
	MV540H_F,
	MV540H_H,
	MV560U_F,
	MV560U_H,
	V430F	(*Omron*)

);
END_TYPE

// ---- DUTs/METS/Device/Scanner/E_SCANNER_State.TcDUT
{attribute 'qualified_only'}
{attribute 'strict'}
TYPE E_SCANNER_State :
(
	IDLE,
	CONNECT,
	SEND,
	RECEIVE,
	DISCONNECT,
	CHECKOS,
	BROWSE,
	IMAGE,
	DECODE,
	HEARTBEAT,
	DONE
);
END_TYPE

// ---- DUTs/METS/Device/Scanner/E_SCANNER_Vendor.TcDUT
{attribute 'qualified_only'}
{attribute 'strict'}
TYPE E_SCANNER_Vendor :
(
	SIEMENS		:= 1,
	MICROSCAN	:= 2,
	OMRON 		:= 3,
	KEYENCE		:= 4,
	COGNEX		:= 5
);
END_TYPE

// ---- DUTs/METS/Device/Scanner/Hand Scanner/E_DataSequence.TcDUT
{attribute 'qualified_only'}
{attribute 'strict'}
TYPE E_DataSequence :
(	
	//E_Send,
	//E_SendWait,
	//E_Recieve,
	//E_RecieveWait
	DUMMY
);
END_TYPE

// ---- DUTs/METS/Device/Scanner/Hand Scanner/ST_SCANNER_HoneywellConfig.TcDUT
TYPE ST_SCANNER_HoneywellConfig :
STRUCT
	bEnabled					: BOOL;										(* Enable HandScanner *)
	sDeviceName				: STRING(30) := 'HandScanner';
	bReset					: BOOL;										(* Reset HandScanner *)
	nScannerPosition			: UINT;										(* Array position used in the camera configs.  This allows the HMi to display the handscanner stuff as a microscan camera *)
	eComPortMode			: ComSerialLineMode_t := SERIALLINEMODE_EL6_22B;	(* COM port type, PC/KL/EL COM ports can all be used - SERIALLINEMODE_EL6_22B *)
	nBaudRate				: UDINT:= 115200;								(* Baud rate for scanner. 2 = 1200, 3=2400, 4=4800, 5=9600, 6=19200, 7=38400, 8=57600, 9=115200 - Default baudrate for hand sanner sick1910i *)
  	nDatabits      				: BYTE := 8;             								(*  8   *)
  	eParity          				: ComParity_t;      								(* PARITY_NONE=0*)
  	nStopbits             			: BYTE := 1;            								 (* 1  *)
	tRXTimeOut				: TIME := T#0ms;
	sReplacmentChar			: T_Char  := '';
END_STRUCT
END_TYPE

// ---- DUTs/METS/Device/Scanner/Hand Scanner/ST_SCANNER_HoneywellCtrl.TcDUT
TYPE ST_SCANNER_HoneywellCtrl :
STRUCT
	bEnableAck							: BOOL;
	bTrigger						: BOOL;
	bResetTirgger					: BOOL;
	bReset							: BOOL;
	bBeepOn						: BOOL;
	bBeepOff						: BOOL;
	bPowerUpBeepOff				: BOOL;
	bPowerUpBeepOn				: BOOL;
	(*bHealth							: BOOL;*)
	bInfo							: BOOL;
	(*bNotOnFile						: BOOL;*)
	(*stHostAck						: ST_SCANNER_HostAck;*)

(*	nState							: BYTE;
	bResetStats						: BOOL;
	sSStats_Pack					: ST_SCANNER_Statistics;
	sSStats_Carton					: ST_SCANNER_Statistics;
	sSStats_Case					: ST_SCANNER_Statistics;
	sCameraEvaluation				:  ST_SCANNER_Evaluation; (* copied in and out of nvram *)

	UID								: UINT;

(* Outputs *)
	strStringReceived				: STRING(255);
	bStringReceived					: BOOL;
	bError							: BOOL;

	eCodeType						: E_CodeType;
	bPackBarcode					: BOOL;
	bCartonBarcode					: BOOL;
	bCaseBarcode					: BOOL;
	sScannerBarcode				: STRING(255);*)
END_STRUCT
END_TYPE

// ---- DUTs/METS/Device/Scanner/Hand Scanner/ST_SCANNER_HoneywellStatus.TcDUT
TYPE ST_SCANNER_HoneywellStatus :
STRUCT
	bStringReceived			: BOOL;
	bExtStringReceived			: BOOL;
	bHandScanerPortOK			: BOOL;
	bHandScannerBaudrateOK	: BOOL;
	sLastScannerBarcode		: STRING(255);
END_STRUCT
END_TYPE

// ---- DUTs/METS/Device/Scanner/Hand Scanner/ST_SCANNER_HostAck.TcDUT
TYPE ST_SCANNER_HostAck :
STRUCT
	bSetHostAckTimeOut				: BOOL;
	tAckTimeOut						: TIME;
	bGoodReadResponse				: BOOL;
	bBadReadResponse				: BOOL;
END_STRUCT
END_TYPE

